C03659=1172.172,406.681,-85.424,-176.064,9.284,148.745
C03660=1172.175,406.433,-85.388,-176.064,9.282,148.745
C03661=1172.179,406.186,-85.352,-176.063,9.280,148.744
C03662=1172.183,405.938,-85.316,-176.063,9.278,148.744
C03663=1172.187,405.691,-85.279,-176.062,9.276,148.743
C03664=1172.191,405.444,-85.244,-176.062,9.273,148.742
C03665=1172.195,405.197,-85.207,-176.062,9.272,148.742
C03666=1172.199,404.949,-85.171,-176.062,9.269,148.741
C03667=1172.204,404.702,-85.135,-176.062,9.267,148.740
C03668=1172.207,404.455,-85.099,-176.061,9.265,148.740
C03669=1172.211,404.207,-85.063,-176.061,9.263,148.739
C03670=1172.215,403.960,-85.027,-176.061,9.261,148.739
C03671=1172.219,403.713,-84.991,-176.060,9.259,148.738
C03672=1172.223,403.465,-84.955,-176.060,9.257,148.737
C03673=1172.226,403.218,-84.919,-176.060,9.255,148.737
C03674=1172.231,402.970,-84.883,-176.060,9.252,148.736
C03675=1172.234,402.724,-84.846,-176.059,9.250,148.735
C03676=1172.238,402.476,-84.810,-176.059,9.248,148.735
C03677=1172.242,402.228,-84.775,-176.059,9.245,148.734
C03678=1172.246,401.981,-84.738,-176.059,9.244,148.733
C03679=1172.250,401.734,-84.702,-176.058,9.241,148.733
C03680=1172.254,401.486,-84.665,-176.058,9.239,148.732
C03681=1172.258,401.239,-84.630,-176.058,9.237,148.731
C03682=1172.261,400.991,-84.594,-176.057,9.234,148.731
C03683=1172.266,400.745,-84.558,-176.058,9.232,148.730
C03684=1172.270,400.497,-84.522,-176.057,9.230,148.729
C03685=1172.274,400.250,-84.486,-176.057,9.228,148.729
C03686=1172.277,400.003,-84.450,-176.057,9.225,148.728
C03687=1172.282,399.755,-84.414,-176.056,9.222,148.727
C03688=1172.285,399.507,-84.378,-176.056,9.220,148.727
C03689=1172.289,399.260,-84.342,-176.056,9.218,148.726
C03690=1172.293,399.013,-84.306,-176.056,9.216,148.725
C03691=1172.297,398.765,-84.270,-176.056,9.213,148.725
C03692=1172.301,398.518,-84.233,-176.056,9.211,148.724
C03693=1172.305,398.270,-84.198,-176.055,9.208,148.723
C03694=1172.308,398.023,-84.162,-176.055,9.206,148.723
C03695=1172.313,397.776,-84.126,-176.055,9.204,148.722
C03696=1172.317,397.529,-84.090,-176.054,9.201,148.721
C03697=1172.321,397.281,-84.054,-176.054,9.199,148.720
C03698=1172.324,397.034,-84.018,-176.054,9.196,148.720
C03699=1172.328,396.787,-83.982,-176.054,9.194,148.719
C03700=1172.332,396.539,-83.946,-176.054,9.191,148.718
C03701=1172.336,396.291,-83.911,-176.054,9.189,148.718
C03702=1172.340,396.044,-83.874,-176.054,9.186,148.717
C03703=1172.344,395.797,-83.838,-176.054,9.184,148.716
C03704=1172.347,395.549,-83.803,-176.054,9.181,148.716
C03705=1172.352,395.303,-83.766,-176.053,9.179,148.715
C03706=1172.356,395.055,-83.731,-176.053,9.176,148.714
C03707=1172.360,394.807,-83.694,-176.053,9.173,148.713
C03708=1172.364,394.560,-83.659,-176.053,9.171,148.713
C03709=1172.367,394.313,-83.623,-176.053,9.167,148.712
C03710=1172.372,394.065,-83.587,-176.053,9.165,148.711
C03711=1172.375,393.818,-83.551,-176.053,9.162,148.711
C03712=1172.379,393.570,-83.515,-176.053,9.160,148.710
C03713=1172.383,393.323,-83.479,-176.053,9.157,148.709
C03714=1172.387,393.076,-83.443,-176.053,9.155,148.709
C03715=1172.391,392.829,-83.408,-176.053,9.152,148.708
C03716=1172.395,392.581,-83.372,-176.053,9.149,148.707
C03717=1172.399,392.334,-83.335,-176.053,9.146,148.706
C03718=1172.404,392.049,-83.294,-176.053,9.143,148.705
C03719=1172.408,391.765,-83.253,-176.053,9.140,148.705
C03720=1172.412,391.480,-83.212,-176.053,9.137,148.704
C03721=1172.417,391.195,-83.171,-176.053,9.133,148.703
C03722=1172.421,390.948,-83.135,-176.054,9.131,148.702
C03723=1172.425,390.700,-83.099,-176.054,9.127,148.702
C03724=1172.429,390.453,-83.063,-176.054,9.125,148.701
C03725=1172.432,390.205,-83.028,-176.054,9.121,148.700
C03726=1172.437,389.957,-82.992,-176.054,9.119,148.699
C03727=1172.440,389.711,-82.955,-176.055,9.115,148.699
C03728=1172.444,389.463,-82.920,-176.054,9.113,148.698
C03729=1172.449,389.216,-82.884,-176.055,9.110,148.697
C03730=1172.452,388.968,-82.848,-176.055,9.107,148.697
C03731=1172.456,388.721,-82.813,-176.055,9.104,148.696
C03732=1172.460,388.473,-82.777,-176.055,9.101,148.695
C03733=1172.464,388.226,-82.741,-176.056,9.098,148.694
C03734=1172.468,387.978,-82.706,-176.057,9.095,148.694
C03735=1172.472,387.732,-82.670,-176.056,9.092,148.693
C03736=1172.475,387.484,-82.634,-176.057,9.089,148.692
C03737=1172.480,387.237,-82.598,-176.057,9.085,148.692
C03738=1172.483,386.989,-82.562,-176.058,9.082,148.691
C03739=1172.487,386.742,-82.527,-176.058,9.080,148.690
C03740=1172.491,386.494,-82.491,-176.058,9.076,148.690
C03741=1172.496,386.247,-82.456,-176.059,9.073,148.689
C03742=1172.499,386.000,-82.420,-176.060,9.070,148.688
C03743=1172.503,385.752,-82.385,-176.060,9.067,148.687
C03744=1172.507,385.505,-82.349,-176.061,9.063,148.687
C03745=1172.511,385.257,-82.313,-176.061,9.060,148.686
C03746=1172.515,385.009,-82.277,-176.062,9.057,148.685
C03747=1172.519,384.762,-82.242,-176.062,9.054,148.685
C03748=1172.523,384.515,-82.207,-176.063,9.050,148.684
C03749=1172.526,384.267,-82.171,-176.064,9.047,148.683
C03750=1172.531,384.020,-82.135,-176.064,9.044,148.683
C03751=1172.534,383.772,-82.099,-176.065,9.041,148.682
C03752=1172.539,383.525,-82.064,-176.065,9.037,148.681
C03753=1172.542,383.278,-82.029,-176.066,9.034,148.681
C03754=1172.546,383.030,-81.993,-176.067,9.031,148.680
C03755=1172.550,382.782,-81.957,-176.067,9.028,148.679
C03756=1172.555,382.536,-81.922,-176.068,9.025,148.679
C03757=1172.558,382.288,-81.886,-176.069,9.020,148.678
C03758=1172.562,382.041,-81.851,-176.070,9.017,148.677
C03759=1172.566,381.793,-81.815,-176.071,9.014,148.677
C03760=1172.569,381.546,-81.780,-176.071,9.011,148.676
C03761=1172.574,381.299,-81.744,-176.073,9.007,148.675
C03762=1172.578,381.051,-81.708,-176.074,9.004,148.675
C03763=1172.582,380.804,-81.673,-176.074,9.000,148.674
C03764=1172.586,380.555,-81.638,-176.075,8.997,148.673
C03765=1172.590,380.309,-81.603,-176.076,8.993,148.673
C03766=1172.594,380.061,-81.567,-176.077,8.990,148.672
C03767=1172.597,379.814,-81.532,-176.078,8.986,148.671
C03768=1172.602,379.566,-81.495,-176.079,8.983,148.671
C03769=1172.606,379.319,-81.460,-176.080,8.980,148.670
C03770=1172.610,379.072,-81.425,-176.081,8.976,148.670
C03771=1172.614,378.823,-81.390,-176.082,8.973,148.669
C03772=1172.618,378.577,-81.355,-176.083,8.969,148.668
C03773=1172.621,378.329,-81.319,-176.084,8.966,148.668
C03774=1172.625,378.082,-81.284,-176.086,8.962,148.667
C03775=1172.629,377.834,-81.249,-176.087,8.959,148.667
C03776=1172.633,377.587,-81.214,-176.088,8.955,148.666
C03777=1172.637,377.339,-81.178,-176.089,8.951,148.665
C03778=1172.641,377.092,-81.142,-176.090,8.948,148.665
C03779=1172.645,376.844,-81.108,-176.092,8.944,148.664
C03780=1172.649,376.597,-81.072,-176.092,8.941,148.664
C03781=1172.653,376.349,-81.037,-176.094,8.937,148.663
C03782=1172.657,376.103,-81.002,-176.095,8.933,148.662
C03783=1172.661,375.854,-80.967,-176.097,8.930,148.662
C03784=1172.664,375.607,-80.931,-176.098,8.926,148.661
C03785=1172.668,375.359,-80.896,-176.099,8.923,148.661
C03786=1172.673,375.112,-80.861,-176.100,8.919,148.660
C03787=1172.676,374.864,-80.826,-176.102,8.916,148.660
C03788=1172.680,374.617,-80.790,-176.103,8.912,148.659
C03789=1172.685,374.370,-80.756,-176.105,8.908,148.658
C03790=1172.688,374.122,-80.720,-176.106,8.905,148.658
C03791=1172.692,373.874,-80.685,-176.108,8.901,148.657
C03792=1172.696,373.627,-80.650,-176.109,8.897,148.657
C03793=1172.700,373.380,-80.615,-176.111,8.894,148.656
C03794=1172.705,373.132,-80.580,-176.112,8.890,148.656
C03795=1172.708,372.885,-80.545,-176.114,8.886,148.655
C03796=1172.712,372.637,-80.510,-176.115,8.883,148.655
C03797=1172.717,372.390,-80.475,-176.117,8.880,148.654
C03798=1172.721,372.142,-80.440,-176.118,8.876,148.654
C03799=1172.724,371.894,-80.404,-176.120,8.872,148.653
C03800=1172.729,371.647,-80.370,-176.121,8.868,148.653
C03801=1172.732,371.400,-80.335,-176.123,8.864,148.652
C03802=1172.736,371.152,-80.300,-176.125,8.861,148.651
C03803=1172.740,370.905,-80.265,-176.126,8.857,148.651
C03804=1172.744,370.656,-80.230,-176.128,8.853,148.651
C03805=1172.748,370.410,-80.195,-176.130,8.849,148.650
C03806=1172.752,370.162,-80.160,-176.132,8.846,148.650
C03807=1172.757,369.914,-80.125,-176.133,8.842,148.649
C03808=1172.760,369.667,-80.090,-176.135,8.839,148.649
C03809=1172.764,369.419,-80.056,-176.137,8.835,148.648
C03810=1172.768,369.172,-80.021,-176.138,8.831,148.648
C03811=1172.772,368.924,-79.986,-176.140,8.827,148.647
C03812=1172.776,368.677,-79.951,-176.142,8.824,148.647
C03813=1172.780,368.429,-79.916,-176.144,8.820,148.646
C03814=1172.784,368.182,-79.882,-176.146,8.817,148.646
C03815=1172.788,367.934,-79.847,-176.148,8.813,148.646
C03816=1172.792,367.686,-79.811,-176.150,8.809,148.645
C03817=1172.796,367.439,-79.777,-176.151,8.806,148.645
C03818=1172.800,367.191,-79.742,-176.153,8.802,148.644
C03819=1172.804,366.944,-79.708,-176.155,8.799,148.644
C03820=1172.808,366.696,-79.673,-176.157,8.795,148.643
C03821=1172.812,366.449,-79.638,-176.159,8.791,148.643
C03822=1172.816,366.166,-79.598,-176.161,8.787,148.642
C03823=1172.821,365.885,-79.559,-176.164,8.783,148.642
C03824=1172.825,365.603,-79.520,-176.166,8.778,148.641
C03825=1172.830,365.321,-79.480,-176.168,8.774,148.641
C03826=1172.834,365.073,-79.445,-176.170,8.771,148.641
C03827=1172.838,364.826,-79.411,-176.172,8.766,148.640
C03828=1172.842,364.578,-79.377,-176.174,8.763,148.640
C03829=1172.846,364.330,-79.342,-176.176,8.759,148.639
C03830=1172.850,364.082,-79.307,-176.178,8.756,148.639
C03831=1172.854,363.835,-79.274,-176.180,8.752,148.639
C03832=1172.858,363.588,-79.238,-176.182,8.748,148.638
C03833=1172.861,363.340,-79.204,-176.185,8.745,148.638
C03834=1172.866,363.093,-79.170,-176.186,8.741,148.638
C03835=1172.870,362.845,-79.135,-176.188,8.737,148.637
C03836=1172.874,362.598,-79.101,-176.191,8.734,148.637
C03837=1172.878,362.350,-79.066,-176.193,8.730,148.636
C03838=1172.882,362.103,-79.032,-176.195,8.726,148.636
C03839=1172.886,361.854,-78.997,-176.197,8.723,148.636
C03840=1172.890,361.607,-78.963,-176.199,8.719,148.635
C03841=1172.893,361.359,-78.929,-176.201,8.716,148.635
C03842=1172.898,361.112,-78.894,-176.204,8.711,148.635
C03843=1172.902,360.865,-78.860,-176.206,8.708,148.634
C03844=1172.906,360.617,-78.826,-176.208,8.704,148.634
C03845=1172.910,360.369,-78.792,-176.210,8.701,148.634
C03846=1172.913,360.121,-78.757,-176.212,8.697,148.633
C03847=1172.918,359.874,-78.724,-176.215,8.693,148.633
C03848=1172.922,359.626,-78.689,-176.217,8.690,148.633
C03849=1172.925,359.378,-78.655,-176.219,8.686,148.632
C03850=1172.930,359.131,-78.621,-176.221,8.682,148.632
C03851=1172.933,358.883,-78.586,-176.223,8.679,148.632
C03852=1172.938,358.636,-78.552,-176.225,8.675,148.631
C03853=1172.942,358.388,-78.519,-176.228,8.672,148.631
C03854=1172.946,358.140,-78.484,-176.230,8.668,148.631
C03855=1172.950,357.893,-78.450,-176.232,8.664,148.630
C03856=1172.954,357.645,-78.416,-176.235,8.661,148.630
C03857=1172.958,357.398,-78.381,-176.237,8.657,148.630
C03858=1172.962,357.149,-78.348,-176.239,8.653,148.629
C03859=1172.966,356.902,-78.314,-176.242,8.650,148.629
C03860=1172.969,356.655,-78.279,-176.244,8.646,148.629
C03861=1172.974,356.407,-78.245,-176.246,8.643,148.629
C03862=1172.978,356.159,-78.212,-176.248,8.640,148.628
C03863=1172.982,355.911,-78.177,-176.251,8.635,148.628
C03864=1172.986,355.664,-78.143,-176.253,8.632,148.628
C03865=1172.990,355.416,-78.110,-176.255,8.628,148.627
C03866=1172.994,355.168,-78.075,-176.257,8.625,148.627
C03867=1172.998,354.921,-78.042,-176.260,8.621,148.627
C03868=1173.002,354.674,-78.008,-176.262,8.617,148.627
C03869=1173.007,354.426,-77.974,-176.264,8.614,148.626
C03870=1173.010,354.178,-77.940,-176.266,8.611,148.626
C03871=1173.014,353.931,-77.906,-176.269,8.607,148.626
C03872=1173.019,353.683,-77.872,-176.271,8.603,148.625
C03873=1173.023,353.435,-77.839,-176.273,8.600,148.625
C03874=1173.026,353.187,-77.805,-176.276,8.597,148.625
C03875=1173.031,352.940,-77.771,-176.278,8.593,148.625
C03876=1173.035,352.692,-77.737,-176.281,8.589,148.624
C03877=1173.039,352.445,-77.704,-176.283,8.585,148.624
C03878=1173.042,352.196,-77.670,-176.285,8.582,148.624
C03879=1173.047,351.949,-77.636,-176.287,8.579,148.624
C03880=1173.051,351.701,-77.602,-176.289,8.576,148.623
C03881=1173.055,351.454,-77.569,-176.292,8.571,148.623
C03882=1173.058,351.206,-77.535,-176.295,8.568,148.623
C03883=1173.063,350.958,-77.501,-176.296,8.565,148.622
C03884=1173.067,350.710,-77.467,-176.299,8.561,148.622
C03885=1173.071,350.463,-77.434,-176.301,8.558,148.622
C03886=1173.075,350.216,-77.400,-176.304,8.554,148.622
C03887=1173.079,349.967,-77.367,-176.306,8.550,148.622
C03888=1173.083,349.719,-77.333,-176.308,8.547,148.621
C03889=1173.087,349.472,-77.299,-176.311,8.544,148.621
C03890=1173.091,349.224,-77.266,-176.313,8.541,148.621
C03891=1173.096,348.977,-77.233,-176.315,8.536,148.620
C03892=1173.099,348.729,-77.199,-176.318,8.533,148.620
C03893=1173.103,348.481,-77.166,-176.320,8.530,148.620
C03894=1173.108,348.233,-77.132,-176.322,8.526,148.620
C03895=1173.112,347.985,-77.099,-176.324,8.523,148.620
C03896=1173.116,347.738,-77.065,-176.327,8.519,148.619
C03897=1173.120,347.490,-77.032,-176.330,8.515,148.619
C03898=1173.124,347.243,-76.998,-176.332,8.512,148.619
C03899=1173.128,346.995,-76.965,-176.334,8.509,148.619
C03900=1173.132,346.747,-76.932,-176.336,8.506,148.618
C03901=1173.136,346.499,-76.898,-176.339,8.502,148.618
C03902=1173.140,346.252,-76.865,-176.342,8.498,148.618
C03903=1173.144,346.004,-76.832,-176.344,8.495,148.618
C03904=1173.148,345.756,-76.798,-176.346,8.492,148.618
C03905=1173.153,345.508,-76.765,-176.348,8.488,148.617
C03906=1173.157,345.260,-76.732,-176.351,8.485,148.617
C03907=1173.161,345.013,-76.698,-176.353,8.482,148.617
C03908=1173.165,344.765,-76.665,-176.356,8.478,148.617
C03909=1173.169,344.517,-76.632,-176.358,8.474,148.616
C03910=1173.174,344.270,-76.599,-176.360,8.471,148.616
C03911=1173.178,344.022,-76.566,-176.363,8.468,148.616
C03912=1173.181,343.773,-76.532,-176.365,8.464,148.616
C03913=1173.185,343.526,-76.499,-176.367,8.461,148.616
C03914=1173.190,343.278,-76.466,-176.370,8.457,148.615
C03915=1173.194,343.030,-76.433,-176.372,8.454,148.615
C03916=1173.198,342.782,-76.400,-176.375,8.450,148.615
C03917=1173.201,342.535,-76.367,-176.377,8.447,148.615
C03918=1173.205,342.287,-76.334,-176.379,8.444,148.614
C03919=1173.209,342.040,-76.301,-176.382,8.441,148.614
C03920=1173.214,341.792,-76.268,-176.384,8.437,148.614
C03921=1173.218,341.544,-76.234,-176.387,8.433,148.614
C03922=1173.222,341.296,-76.201,-176.389,8.430,148.614
C03923=1173.226,341.049,-76.168,-176.392,8.427,148.614
C03924=1173.230,340.801,-76.135,-176.394,8.423,148.613
C03925=1173.235,340.553,-76.103,-176.396,8.420,148.613
C03926=1173.239,340.274,-76.066,-176.399,8.416,148.613
C03927=1173.244,339.994,-76.028,-176.402,8.412,148.613
C03928=1173.248,339.715,-75.991,-176.405,8.409,148.613
C03929=1173.253,339.436,-75.954,-176.407,8.405,148.612
C03930=1173.257,339.189,-75.921,-176.410,8.401,148.612
C03931=1173.261,338.940,-75.889,-176.412,8.398,148.612
C03932=1173.265,338.693,-75.856,-176.414,8.395,148.612
C03933=1173.270,338.445,-75.822,-176.416,8.391,148.612
C03934=1173.273,338.197,-75.790,-176.419,8.388,148.612
C03935=1173.277,337.949,-75.757,-176.422,8.384,148.611
C03936=1173.282,337.701,-75.724,-176.424,8.381,148.611
C03937=1173.286,337.454,-75.691,-176.427,8.378,148.611
C03938=1173.289,337.206,-75.659,-176.429,8.374,148.611
C03939=1173.294,336.958,-75.626,-176.431,8.371,148.610
C03940=1173.298,336.709,-75.594,-176.434,8.368,148.610
C03941=1173.303,336.462,-75.561,-176.436,8.365,148.610
C03942=1173.306,336.215,-75.528,-176.438,8.362,148.610
C03943=1173.311,335.967,-75.496,-176.441,8.357,148.610
C03944=1173.315,335.719,-75.463,-176.444,8.354,148.610
C03945=1173.318,335.471,-75.431,-176.446,8.351,148.610
C03946=1173.323,335.223,-75.398,-176.449,8.348,148.609
C03947=1173.327,334.975,-75.365,-176.451,8.344,148.609
C03948=1173.331,334.727,-75.332,-176.453,8.341,148.609
C03949=1173.335,334.480,-75.300,-176.456,8.338,148.609
C03950=1173.340,334.232,-75.267,-176.458,8.335,148.609
C03951=1173.343,333.985,-75.235,-176.460,8.332,148.609
C03952=1173.347,333.736,-75.202,-176.463,8.327,148.608
C03953=1173.352,333.488,-75.170,-176.466,8.324,148.608
C03954=1173.355,333.240,-75.137,-176.468,8.321,148.608
C03955=1173.360,332.992,-75.105,-176.471,8.318,148.608
C03956=1173.364,332.744,-75.072,-176.473,8.315,148.608
C03957=1173.368,332.497,-75.040,-176.476,8.312,148.608
C03958=1173.373,332.249,-75.008,-176.478,8.308,148.607
C03959=1173.376,332.001,-74.975,-176.480,8.305,148.607
C03960=1173.380,331.753,-74.943,-176.483,8.302,148.607
C03961=1173.384,331.506,-74.910,-176.485,8.299,148.607
C03962=1173.389,331.258,-74.878,-176.487,8.295,148.607
C03963=1173.393,331.010,-74.846,-176.491,8.292,148.607
C03964=1173.397,330.762,-74.813,-176.493,8.288,148.607
C03965=1173.401,330.514,-74.781,-176.495,8.285,148.606
C03966=1173.405,330.266,-74.749,-176.498,8.282,148.606
C03967=1173.410,330.018,-74.717,-176.500,8.279,148.606
C03968=1173.413,329.771,-74.684,-176.503,8.275,148.606
C03969=1173.418,329.522,-74.652,-176.505,8.272,148.606
C03970=1173.421,329.274,-74.620,-176.508,8.269,148.606
C03971=1173.427,329.027,-74.588,-176.510,8.266,148.606
C03972=1173.430,328.779,-74.556,-176.513,8.263,148.606
C03973=1173.434,328.531,-74.523,-176.515,8.259,148.605
C03974=1173.438,328.283,-74.491,-176.517,8.256,148.605
C03975=1173.442,328.035,-74.460,-176.520,8.252,148.605
C03976=1173.447,327.787,-74.427,-176.523,8.249,148.605
C03977=1173.451,327.539,-74.395,-176.525,8.246,148.605
C03978=1173.455,327.291,-74.363,-176.528,8.243,148.605
C03979=1173.459,327.043,-74.332,-176.530,8.239,148.605
C03980=1173.463,326.796,-74.299,-176.532,8.236,148.604
C03981=1173.467,326.548,-74.267,-176.535,8.233,148.604
C03982=1173.471,326.300,-74.235,-176.537,8.230,148.604
C03983=1173.476,326.052,-74.203,-176.540,8.227,148.604
C03984=1173.480,325.804,-74.171,-176.542,8.224,148.604
C03985=1173.484,325.557,-74.139,-176.544,8.220,148.604
C03986=1173.488,325.308,-74.107,-176.547,8.217,148.604
C03987=1173.492,325.060,-74.075,-176.549,8.214,148.604
C03988=1173.496,324.812,-74.043,-176.552,8.211,148.604
C03989=1173.501,324.564,-74.011,-176.554,8.208,148.603
C03990=1173.505,324.316,-73.979,-176.557,8.204,148.603
C03991=1173.508,324.068,-73.947,-176.560,8.201,148.603
C03992=1173.513,323.821,-73.916,-176.562,8.197,148.603
C03993=1173.517,323.572,-73.884,-176.565,8.194,148.603
C03994=1173.522,323.325,-73.853,-176.567,8.191,148.603
C03995=1173.525,323.077,-73.821,-176.570,8.188,148.603
C03996=1173.530,322.828,-73.788,-176.572,8.185,148.602
C03997=1173.534,322.581,-73.757,-176.575,8.181,148.602
C03998=1173.538,322.333,-73.725,-176.577,8.178,148.602
C03999=1173.541,322.085,-73.693,-176.580,8.175,148.602
C04000=1173.546,321.837,-73.662,-176.582,8.172,148.602
C04001=1173.551,321.589,-73.630,-176.585,8.169,148.602
C04002=1173.555,321.341,-73.599,-176.587,8.166,148.602
C04003=1173.559,321.093,-73.567,-176.590,8.163,148.602
C04004=1173.562,320.845,-73.535,-176.592,8.160,148.602
C04005=1173.567,320.597,-73.504,-176.595,8.156,148.602
C04006=1173.571,320.349,-73.472,-176.597,8.153,148.602
C04007=1173.576,320.102,-73.440,-176.600,8.150,148.601
C04008=1173.579,319.854,-73.408,-176.602,8.147,148.601
C04009=1173.583,319.605,-73.377,-176.605,8.144,148.601
C04010=1173.588,319.358,-73.346,-176.607,8.141,148.601
C04011=1173.591,319.109,-73.314,-176.610,8.137,148.601
C04012=1173.596,318.862,-73.283,-176.612,8.134,148.601
C04013=1173.600,318.613,-73.251,-176.615,8.131,148.601
C04014=1173.605,318.366,-73.219,-176.617,8.128,148.601
C04015=1173.609,318.117,-73.188,-176.620,8.125,148.601
C04016=1173.613,317.870,-73.157,-176.622,8.122,148.601
C04017=1173.617,317.621,-73.125,-176.625,8.118,148.600
C04018=1173.621,317.374,-73.094,-176.628,8.115,148.600
C04019=1173.625,317.126,-73.062,-176.630,8.111,148.600
C04020=1173.630,316.878,-73.031,-176.633,8.108,148.600
C04021=1173.633,316.630,-73.000,-176.635,8.105,148.600
C04022=1173.638,316.382,-72.969,-176.638,8.102,148.600
C04023=1173.642,316.134,-72.937,-176.640,8.099,148.600
C04024=1173.646,315.886,-72.906,-176.643,8.096,148.600
C04025=1173.650,315.638,-72.874,-176.645,8.093,148.600
C04026=1173.655,315.390,-72.844,-176.648,8.090,148.600
C04027=1173.658,315.142,-72.812,-176.650,8.086,148.599
C04028=1173.663,314.894,-72.781,-176.653,8.083,148.599
C04029=1173.667,314.645,-72.750,-176.655,8.080,148.599
C04030=1173.672,314.368,-72.715,-176.658,8.077,148.599
C04031=1173.676,314.092,-72.680,-176.661,8.073,148.599
C04032=1173.681,313.815,-72.645,-176.664,8.070,148.599
C04033=1173.686,313.538,-72.610,-176.667,8.066,148.599
C04034=1173.690,313.291,-72.579,-176.670,8.063,148.599
C04035=1173.694,313.042,-72.548,-176.672,8.060,148.599
C04036=1173.698,312.794,-72.517,-176.675,8.057,148.599
C04037=1173.702,312.546,-72.486,-176.677,8.053,148.599
C04038=1173.707,312.298,-72.455,-176.680,8.050,148.599
C04039=1173.711,312.050,-72.424,-176.682,8.047,148.598
C04040=1173.715,311.802,-72.392,-176.685,8.044,148.599
C04041=1173.720,311.554,-72.361,-176.687,8.041,148.599
C04042=1173.724,311.305,-72.330,-176.690,8.038,148.598
C04043=1173.728,311.058,-72.300,-176.692,8.035,148.598
C04044=1173.732,310.810,-72.269,-176.695,8.032,148.598
C04045=1173.736,310.562,-72.237,-176.697,8.029,148.598
C04046=1173.740,310.314,-72.207,-176.700,8.026,148.598
C04047=1173.745,310.066,-72.176,-176.702,8.023,148.598
C04048=1173.749,309.817,-72.145,-176.705,8.020,148.598
C04049=1173.753,309.570,-72.115,-176.707,8.017,148.598
C04050=1173.757,309.321,-72.083,-176.710,8.014,148.598
C04051=1173.761,309.074,-72.052,-176.712,8.011,148.598
C04052=1173.766,308.826,-72.021,-176.715,8.008,148.598
C04053=1173.770,308.577,-71.990,-176.717,8.005,148.598
C04054=1173.774,308.329,-71.960,-176.720,8.001,148.598
C04055=1173.778,308.081,-71.929,-176.722,7.998,148.598
C04056=1173.782,307.833,-71.898,-176.725,7.995,148.598
C04057=1173.787,307.585,-71.867,-176.727,7.992,148.597
C04058=1173.791,307.337,-71.837,-176.730,7.989,148.597
C04059=1173.796,307.089,-71.806,-176.733,7.986,148.597
C04060=1173.800,306.840,-71.775,-176.735,7.983,148.597
C04061=1173.804,306.592,-71.745,-176.738,7.980,148.597
C04062=1173.808,306.345,-71.714,-176.741,7.977,148.597
C04063=1173.812,306.096,-71.683,-176.743,7.974,148.597
C04064=1173.817,305.848,-71.652,-176.746,7.971,148.597
C04065=1173.821,305.601,-71.622,-176.748,7.968,148.597
C04066=1173.825,305.353,-71.592,-176.751,7.964,148.597
C04067=1173.829,305.104,-71.560,-176.753,7.961,148.597
C04068=1173.833,304.856,-71.530,-176.756,7.958,148.597
C04069=1173.838,304.608,-71.499,-176.758,7.955,148.597
C04070=1173.842,304.360,-71.469,-176.761,7.952,148.597
C04071=1173.846,304.111,-71.439,-176.764,7.949,148.597
C04072=1173.850,303.863,-71.408,-176.766,7.946,148.597
C04073=1173.854,303.616,-71.378,-176.769,7.943,148.597
C04074=1173.859,303.368,-71.347,-176.772,7.940,148.597
C04075=1173.864,303.120,-71.316,-176.774,7.936,148.597
C04076=1173.867,302.872,-71.286,-176.777,7.933,148.597
C04077=1173.872,302.623,-71.256,-176.779,7.931,148.597
C04078=1173.876,302.375,-71.226,-176.781,7.928,148.596
C04079=1173.880,302.127,-71.195,-176.784,7.925,148.596
C04080=1173.885,301.879,-71.164,-176.786,7.922,148.596
C04081=1173.888,301.630,-71.134,-176.789,7.919,148.596
C04082=1173.893,301.382,-71.104,-176.791,7.916,148.596
C04083=1173.897,301.135,-71.073,-176.794,7.913,148.596
C04084=1173.902,300.886,-71.043,-176.797,7.910,148.596
C04085=1173.906,300.639,-71.013,-176.799,7.907,148.596
C04086=1173.910,300.390,-70.982,-176.802,7.904,148.596
C04087=1173.914,300.142,-70.953,-176.805,7.901,148.596
C04088=1173.918,299.894,-70.922,-176.807,7.897,148.596
C04089=1173.922,299.646,-70.892,-176.810,7.894,148.596
C04090=1173.927,299.397,-70.862,-176.812,7.891,148.596
C04091=1173.931,299.150,-70.831,-176.815,7.888,148.596
C04092=1173.935,298.902,-70.802,-176.817,7.885,148.596
C04093=1173.939,298.653,-70.771,-176.820,7.883,148.596
C04094=1173.943,298.405,-70.741,-176.822,7.880,148.596
C04095=1173.948,298.157,-70.711,-176.825,7.877,148.596
C04096=1173.952,297.909,-70.680,-176.827,7.874,148.596
C04097=1173.957,297.660,-70.650,-176.830,7.871,148.596
C04098=1173.961,297.413,-70.620,-176.833,7.868,148.596
C04099=1173.965,297.165,-70.591,-176.836,7.865,148.596
C04100=1173.970,296.917,-70.560,-176.838,7.861,148.596
C04101=1173.974,296.668,-70.531,-176.841,7.858,148.596
C04102=1173.978,296.421,-70.500,-176.843,7.855,148.596
C04103=1173.982,296.171,-70.470,-176.846,7.852,148.596
C04104=1173.986,295.923,-70.441,-176.848,7.849,148.596
C04105=1173.990,295.675,-70.410,-176.851,7.846,148.596
C04106=1173.995,295.427,-70.380,-176.853,7.844,148.596
C04107=1173.999,295.179,-70.350,-176.856,7.841,148.596
C04108=1174.003,294.931,-70.321,-176.858,7.838,148.596
C04109=1174.008,294.682,-70.291,-176.861,7.835,148.596
C04110=1174.012,294.435,-70.260,-176.864,7.832,148.596
C04111=1174.016,294.186,-70.231,-176.866,7.829,148.596
C04112=1174.020,293.938,-70.202,-176.869,7.825,148.595
C04113=1174.025,293.690,-70.171,-176.871,7.822,148.596
C04114=1174.029,293.442,-70.141,-176.874,7.819,148.596
C04115=1174.033,293.194,-70.112,-176.877,7.817,148.596
C04116=1174.037,292.946,-70.082,-176.879,7.814,148.596
C04117=1174.042,292.698,-70.052,-176.881,7.811,148.595
C04118=1174.046,292.449,-70.022,-176.884,7.808,148.596
C04119=1174.050,292.201,-69.993,-176.887,7.805,148.596
C04120=1174.055,291.953,-69.963,-176.890,7.802,148.596
C04121=1174.058,291.705,-69.933,-176.892,7.799,148.596
C04122=1174.063,291.456,-69.903,-176.895,7.796,148.595
C04123=1174.067,291.208,-69.874,-176.897,7.793,148.595
C04124=1174.072,290.960,-69.844,-176.900,7.790,148.595
C04125=1174.076,290.712,-69.815,-176.903,7.787,148.596
C04126=1174.080,290.463,-69.785,-176.905,7.785,148.596
C04127=1174.084,290.216,-69.755,-176.908,7.782,148.596
C04128=1174.089,289.967,-69.725,-176.910,7.778,148.595
C04129=1174.093,289.719,-69.696,-176.913,7.775,148.595
C04130=1174.097,289.471,-69.666,-176.915,7.773,148.596
C04131=1174.101,289.222,-69.637,-176.918,7.770,148.596
C04132=1174.106,288.974,-69.607,-176.921,7.767,148.596
C04133=1174.110,288.726,-69.578,-176.923,7.763,148.595
C04134=1174.115,288.452,-69.545,-176.926,7.760,148.595
C04135=1174.119,288.177,-69.513,-176.929,7.757,148.595
C04136=1174.124,287.901,-69.480,-176.931,7.754,148.595
C04137=1174.129,287.627,-69.447,-176.935,7.751,148.595
C04138=1174.134,287.379,-69.418,-176.937,7.748,148.596
C04139=1174.138,287.131,-69.388,-176.940,7.745,148.596
C04140=1174.142,286.882,-69.359,-176.942,7.742,148.596
C04141=1174.146,286.634,-69.329,-176.945,7.739,148.596
C04142=1174.150,286.386,-69.300,-176.947,7.736,148.595
C04143=1174.154,286.138,-69.271,-176.950,7.733,148.596
C04144=1174.159,285.889,-69.242,-176.953,7.730,148.596
C04145=1174.164,285.641,-69.213,-176.956,7.727,148.596
C04146=1174.168,285.393,-69.183,-176.958,7.725,148.596
C04147=1174.172,285.145,-69.154,-176.960,7.722,148.596
C04148=1174.176,284.896,-69.124,-176.963,7.719,148.596
C04149=1174.180,284.648,-69.095,-176.966,7.716,148.596
C04150=1174.185,284.399,-69.066,-176.968,7.713,148.596
C04151=1174.190,284.152,-69.037,-176.971,7.710,148.596
C04152=1174.194,283.903,-69.008,-176.974,7.707,148.596
C04153=1174.198,283.655,-68.978,-176.976,7.705,148.596
C04154=1174.202,283.407,-68.949,-176.979,7.702,148.596
C04155=1174.206,283.158,-68.921,-176.981,7.699,148.596
C04156=1174.210,282.910,-68.891,-176.984,7.696,148.596
C04157=1174.215,282.662,-68.862,-176.987,7.693,148.596
C04158=1174.219,282.414,-68.833,-176.990,7.690,148.596
C04159=1174.224,282.165,-68.804,-176.992,7.687,148.596
C04160=1174.228,281.917,-68.774,-176.994,7.684,148.596
C04161=1174.233,281.670,-68.745,-176.997,7.681,148.596
C04162=1174.237,281.421,-68.717,-176.999,7.678,148.596
C04163=1174.241,281.173,-68.688,-177.002,7.675,148.596
C04164=1174.245,280.924,-68.659,-177.005,7.672,148.596
C04165=1174.250,280.676,-68.630,-177.008,7.669,148.596
C04166=1174.254,280.428,-68.600,-177.010,7.667,148.596
C04167=1174.258,280.179,-68.572,-177.013,7.664,148.596
C04168=1174.263,279.931,-68.542,-177.015,7.661,148.596
C04169=1174.267,279.683,-68.514,-177.018,7.658,148.596
C04170=1174.271,279.435,-68.485,-177.021,7.655,148.596
C04171=1174.275,279.186,-68.456,-177.022,7.653,148.596
C04172=1174.280,278.937,-68.427,-177.025,7.650,148.596
C04173=1174.284,278.690,-68.398,-177.028,7.647,148.596
C04174=1174.288,278.441,-68.370,-177.031,7.644,148.596
C04175=1174.293,278.193,-68.340,-177.033,7.641,148.596
C04176=1174.297,277.944,-68.311,-177.036,7.638,148.596
C04177=1174.301,277.697,-68.283,-177.038,7.636,148.596
C04178=1174.306,277.448,-68.254,-177.041,7.633,148.596
C04179=1174.310,277.199,-68.225,-177.044,7.630,148.597
C04180=1174.314,276.952,-68.197,-177.047,7.627,148.597
C04181=1174.319,276.703,-68.168,-177.049,7.624,148.597
C04182=1174.323,276.455,-68.139,-177.051,7.622,148.597
C04183=1174.327,276.207,-68.111,-177.054,7.619,148.597
C04184=1174.332,275.958,-68.082,-177.057,7.616,148.597
C04185=1174.336,275.710,-68.053,-177.060,7.613,148.597
C04186=1174.340,275.462,-68.025,-177.062,7.610,148.597
C04187=1174.345,275.213,-67.996,-177.065,7.608,148.597
C04188=1174.349,274.965,-67.967,-177.067,7.605,148.597
C04189=1174.353,274.717,-67.939,-177.070,7.602,148.597
C04190=1174.358,274.468,-67.910,-177.073,7.599,148.597
C04191=1174.361,274.220,-67.881,-177.076,7.596,148.597
C04192=1174.366,273.972,-67.853,-177.078,7.594,148.597
C04193=1174.371,273.723,-67.824,-177.080,7.591,148.597
C04194=1174.375,273.475,-67.797,-177.083,7.588,148.597
C04195=1174.379,273.227,-67.767,-177.086,7.585,148.597
C04196=1174.383,272.978,-67.739,-177.089,7.582,148.597
C04197=1174.388,272.730,-67.711,-177.091,7.580,148.597
C04198=1174.392,272.481,-67.682,-177.094,7.577,148.598
C04199=1174.397,272.233,-67.654,-177.096,7.574,148.598
C04200=1174.400,271.985,-67.625,-177.099,7.571,148.598
C04201=1174.405,271.737,-67.597,-177.101,7.569,148.598
C04202=1174.409,271.489,-67.569,-177.104,7.566,148.598
C04203=1174.414,271.240,-67.540,-177.107,7.563,148.598
C04204=1174.418,270.992,-67.512,-177.109,7.560,148.598
C04205=1174.422,270.743,-67.483,-177.112,7.557,148.598
C04206=1174.427,270.495,-67.456,-177.114,7.555,148.598
C04207=1174.431,270.246,-67.427,-177.117,7.552,148.598
C04208=1174.435,269.999,-67.398,-177.120,7.549,148.598
C04209=1174.440,269.750,-67.370,-177.123,7.546,148.598
C04210=1174.444,269.502,-67.342,-177.125,7.544,148.598
C04211=1174.449,269.253,-67.313,-177.128,7.541,148.598
C04212=1174.453,269.005,-67.285,-177.130,7.538,148.598
C04213=1174.458,268.756,-67.257,-177.133,7.535,148.598
C04214=1174.462,268.509,-67.229,-177.135,7.532,148.598
C04215=1174.466,268.260,-67.201,-177.138,7.530,148.598
C04216=1174.471,268.012,-67.172,-177.141,7.527,148.599
C04217=1174.475,267.763,-67.145,-177.143,7.524,148.599
C04218=1174.480,267.514,-67.117,-177.146,7.521,148.599
C04219=1174.484,267.266,-67.088,-177.148,7.518,148.599
C04220=1174.488,267.018,-67.061,-177.151,7.515,148.599
C04221=1174.492,266.769,-67.032,-177.154,7.513,148.599
C04222=1174.497,266.521,-67.004,-177.156,7.510,148.599
C04223=1174.501,266.273,-66.976,-177.159,7.507,148.599
C04224=1174.506,266.024,-66.948,-177.161,7.504,148.599
C04225=1174.509,265.776,-66.920,-177.164,7.501,148.599
C04226=1174.514,265.527,-66.892,-177.167,7.500,148.599
C04227=1174.519,265.278,-66.864,-177.170,7.497,148.599
C04228=1174.523,265.031,-66.836,-177.172,7.494,148.599
C04229=1174.527,264.783,-66.808,-177.175,7.491,148.599
C04230=1174.531,264.534,-66.780,-177.177,7.489,148.600
C04231=1174.536,264.285,-66.752,-177.180,7.486,148.600
C04232=1174.540,264.037,-66.724,-177.183,7.483,148.600
C04233=1174.544,263.789,-66.696,-177.186,7.480,148.600
C04234=1174.550,263.541,-66.668,-177.188,7.478,148.600
C04235=1174.554,263.291,-66.641,-177.190,7.475,148.600
C04236=1174.558,263.044,-66.613,-177.193,7.472,148.600
C04237=1174.562,262.795,-66.585,-177.195,7.469,148.600
C04238=1174.567,262.522,-66.554,-177.199,7.467,148.600
C04239=1174.572,262.249,-66.524,-177.202,7.463,148.600
C04240=1174.576,261.976,-66.493,-177.205,7.460,148.600
C04241=1174.582,261.703,-66.463,-177.207,7.457,148.600
C04242=1174.586,261.454,-66.435,-177.210,7.455,148.601
C04243=1174.590,261.206,-66.408,-177.213,7.452,148.601
C04244=1174.594,260.958,-66.380,-177.215,7.449,148.601
C04245=1174.599,260.709,-66.352,-177.218,7.446,148.601
C04246=1174.603,260.461,-66.324,-177.220,7.444,148.601
C04247=1174.608,260.212,-66.297,-177.223,7.441,148.601
C04248=1174.612,259.964,-66.269,-177.226,7.438,148.601
C04249=1174.617,259.715,-66.242,-177.228,7.436,148.601
C04250=1174.621,259.467,-66.214,-177.231,7.433,148.601
C04251=1174.625,259.218,-66.186,-177.234,7.430,148.602
C04252=1174.629,258.970,-66.159,-177.236,7.428,148.602
C04253=1174.634,258.722,-66.132,-177.239,7.425,148.602
C04254=1174.638,258.473,-66.104,-177.242,7.422,148.602
C04255=1174.643,258.224,-66.076,-177.244,7.419,148.602
C04256=1174.647,257.977,-66.048,-177.247,7.417,148.602
C04257=1174.652,257.728,-66.021,-177.249,7.414,148.602
C04258=1174.656,257.479,-65.993,-177.253,7.412,148.602
C04259=1174.661,257.231,-65.966,-177.255,7.410,148.602
C04260=1174.665,256.982,-65.939,-177.257,7.407,148.602
C04261=1174.669,256.734,-65.911,-177.260,7.404,148.602
C04262=1174.674,256.485,-65.884,-177.262,7.401,148.602
C04263=1174.678,256.238,-65.856,-177.265,7.398,148.603
C04264=1174.683,255.989,-65.829,-177.268,7.396,148.603
C04265=1174.687,255.740,-65.801,-177.271,7.394,148.603
C04266=1174.691,255.492,-65.773,-177.273,7.391,148.603
C04267=1174.696,255.243,-65.746,-177.276,7.388,148.603
C04268=1174.700,254.995,-65.719,-177.278,7.386,148.603
C04269=1174.704,254.746,-65.692,-177.281,7.383,148.603
C04270=1174.709,254.498,-65.664,-177.284,7.380,148.603
C04271=1174.713,254.250,-65.638,-177.286,7.378,148.604
C04272=1174.717,254.001,-65.611,-177.289,7.375,148.604
C04273=1174.722,253.753,-65.584,-177.292,7.372,148.604
C04274=1174.726,253.504,-65.555,-177.294,7.370,148.604
C04275=1174.730,253.256,-65.528,-177.297,7.367,148.604
C04276=1174.735,253.007,-65.501,-177.300,7.364,148.604
C04277=1174.740,252.759,-65.474,-177.302,7.362,148.604
C04278=1174.744,252.510,-65.447,-177.305,7.359,148.604
C04279=1174.749,252.262,-65.420,-177.308,7.356,148.605
C04280=1174.752,252.013,-65.393,-177.310,7.354,148.605
C04281=1174.757,251.765,-65.366,-177.313,7.351,148.605
C04282=1174.761,251.516,-65.338,-177.316,7.348,148.605
C04283=1174.766,251.268,-65.311,-177.318,7.346,148.605
C04284=1174.771,251.019,-65.284,-177.321,7.344,148.605
C04285=1174.775,250.771,-65.257,-177.323,7.341,148.605
C04286=1174.779,250.522,-65.230,-177.326,7.338,148.605
C04287=1174.783,250.274,-65.203,-177.329,7.335,148.605
C04288=1174.788,250.025,-65.176,-177.331,7.334,148.606
C04289=1174.793,249.777,-65.149,-177.334,7.331,148.606
C04290=1174.797,249.528,-65.122,-177.337,7.328,148.606
C04291=1174.801,249.280,-65.096,-177.339,7.326,148.606
C04292=1174.806,249.031,-65.069,-177.342,7.323,148.606
C04293=1174.810,248.783,-65.042,-177.345,7.320,148.606
C04294=1174.815,248.534,-65.014,-177.347,7.318,148.606
C04295=1174.818,248.285,-64.988,-177.350,7.315,148.606
C04296=1174.823,248.037,-64.961,-177.353,7.313,148.607
C04297=1174.828,247.788,-64.934,-177.355,7.310,148.607
C04298=1174.832,247.540,-64.907,-177.358,7.307,148.607
C04299=1174.836,247.292,-64.880,-177.360,7.305,148.607
C04300=1174.841,247.043,-64.853,-177.364,7.302,148.607
C04301=1174.846,246.795,-64.826,-177.366,7.300,148.607
C04302=1174.850,246.546,-64.800,-177.369,7.297,148.607
C04303=1174.855,246.298,-64.773,-177.371,7.294,148.607
C04304=1174.859,246.049,-64.746,-177.374,7.292,148.608
C04305=1174.863,245.801,-64.720,-177.377,7.290,148.608
C04306=1174.868,245.552,-64.693,-177.379,7.287,148.608
C04307=1174.872,245.304,-64.665,-177.382,7.285,148.608
C04308=1174.877,245.055,-64.640,-177.385,7.282,148.608
C04309=1174.881,244.807,-64.613,-177.387,7.280,148.608
C04310=1174.885,244.558,-64.586,-177.390,7.277,148.608
C04311=1174.890,244.310,-64.559,-177.392,7.275,148.609
C04312=1174.895,244.061,-64.533,-177.395,7.272,148.609
C04313=1174.899,243.813,-64.506,-177.398,7.269,148.609
C04314=1174.903,243.564,-64.479,-177.401,7.267,148.609
C04315=1174.907,243.316,-64.453,-177.403,7.264,148.609
C04316=1174.912,243.067,-64.426,-177.405,7.262,148.609
C04317=1174.916,242.819,-64.400,-177.409,7.259,148.610
C04318=1174.921,242.570,-64.373,-177.411,7.256,148.610
C04319=1174.926,242.321,-64.347,-177.414,7.254,148.610
C04320=1174.930,242.073,-64.320,-177.417,7.252,148.610
C04321=1174.935,241.824,-64.294,-177.419,7.250,148.610
C04322=1174.939,241.575,-64.267,-177.422,7.247,148.610
C04323=1174.943,241.327,-64.240,-177.424,7.245,148.611
C04324=1174.948,241.078,-64.214,-177.427,7.242,148.611
C04325=1174.952,240.830,-64.187,-177.430,7.239,148.611
C04326=1174.956,240.581,-64.162,-177.433,7.237,148.611
C04327=1174.961,240.332,-64.135,-177.435,7.234,148.611
C04328=1174.965,240.084,-64.109,-177.437,7.232,148.611
C04329=1174.969,239.835,-64.082,-177.441,7.229,148.612
C04330=1174.974,239.587,-64.055,-177.443,7.227,148.612
C04331=1174.978,239.338,-64.030,-177.446,7.224,148.612
C04332=1174.983,239.090,-64.003,-177.449,7.222,148.612
C04333=1174.988,238.842,-63.977,-177.451,7.219,148.612
C04334=1174.993,238.592,-63.951,-177.454,7.216,148.612
C04335=1174.996,238.344,-63.924,-177.456,7.215,148.612
C04336=1175.001,238.095,-63.899,-177.459,7.212,148.613
C04337=1175.005,237.847,-63.872,-177.462,7.210,148.613
C04338=1175.010,237.598,-63.846,-177.465,7.207,148.613
C04339=1175.014,237.350,-63.819,-177.467,7.205,148.613
C04340=1175.018,237.101,-63.793,-177.470,7.202,148.613
C04341=1175.023,236.853,-63.768,-177.472,7.200,148.613
C04342=1175.028,236.581,-63.738,-177.475,7.197,148.614
C04343=1175.033,236.309,-63.710,-177.478,7.194,148.614
C04344=1175.037,236.038,-63.681,-177.481,7.192,148.614
C04345=1175.043,235.766,-63.653,-177.484,7.189,148.614
C04346=1175.047,235.518,-63.626,-177.486,7.187,148.614
C04347=1175.051,235.269,-63.601,-177.490,7.184,148.615
C04348=1175.057,235.020,-63.575,-177.492,7.182,148.615
C04349=1175.061,234.772,-63.548,-177.495,7.179,148.615
C04350=1175.065,234.523,-63.522,-177.498,7.176,148.615
C04351=1175.069,234.275,-63.497,-177.500,7.174,148.615
C04352=1175.074,234.025,-63.470,-177.503,7.172,148.615
C04353=1175.079,233.777,-63.445,-177.505,7.169,148.616
C04354=1175.083,233.529,-63.418,-177.508,7.167,148.616
C04355=1175.087,233.280,-63.393,-177.511,7.165,148.616
C04356=1175.092,233.031,-63.366,-177.514,7.162,148.616
C04357=1175.096,232.782,-63.341,-177.516,7.160,148.616
C04358=1175.101,232.534,-63.315,-177.519,7.157,148.616
C04359=1175.105,232.286,-63.289,-177.521,7.155,148.617
C04360=1175.110,232.037,-63.262,-177.524,7.152,148.617
C04361=1175.114,231.788,-63.237,-177.527,7.150,148.617
C04362=1175.119,231.540,-63.211,-177.530,7.147,148.617
C04363=1175.123,231.291,-63.185,-177.532,7.146,148.618
C04364=1175.127,231.042,-63.160,-177.535,7.143,148.618
C04365=1175.132,230.794,-63.134,-177.537,7.140,148.618
C04366=1175.137,230.545,-63.108,-177.540,7.138,148.618
C04367=1175.141,230.296,-63.082,-177.543,7.136,148.618
C04368=1175.146,230.048,-63.057,-177.546,7.133,148.618
C04369=1175.150,229.799,-63.031,-177.548,7.131,148.619
C04370=1175.155,229.551,-63.005,-177.551,7.128,148.619
C04371=1175.159,229.302,-62.980,-177.553,7.126,148.619
C04372=1175.163,229.053,-62.954,-177.557,7.124,148.619
C04373=1175.168,228.805,-62.928,-177.559,7.121,148.619
C04374=1175.173,228.556,-62.902,-177.562,7.119,148.620
C04375=1175.177,228.307,-62.876,-177.564,7.117,148.620
C04376=1175.182,228.059,-62.851,-177.567,7.115,148.620
C04377=1175.186,227.810,-62.825,-177.570,7.112,148.620
C04378=1175.190,227.561,-62.799,-177.572,7.110,148.620
C04379=1175.195,227.313,-62.774,-177.575,7.107,148.621
C04380=1175.199,227.064,-62.748,-177.577,7.105,148.621
C04381=1175.204,226.816,-62.723,-177.581,7.102,148.621
C04382=1175.208,226.568,-62.697,-177.583,7.100,148.621
C04383=1175.213,226.318,-62.672,-177.586,7.098,148.621
C04384=1175.217,226.069,-62.646,-177.588,7.096,148.622
C04385=1175.222,225.821,-62.621,-177.591,7.093,148.622
C04386=1175.226,225.572,-62.595,-177.594,7.091,148.622
C04387=1175.230,225.324,-62.570,-177.597,7.088,148.622
C04388=1175.235,225.076,-62.544,-177.599,7.086,148.622
C04389=1175.240,224.826,-62.519,-177.602,7.083,148.623
C04390=1175.244,224.577,-62.493,-177.604,7.081,148.623
C04391=1175.249,224.329,-62.468,-177.607,7.079,148.623
C04392=1175.253,224.080,-62.442,-177.610,7.076,148.623
C04393=1175.258,223.832,-62.418,-177.612,7.075,148.623
C04394=1175.262,223.583,-62.392,-177.615,7.072,148.624
C04395=1175.266,223.334,-62.367,-177.618,7.070,148.624
C04396=1175.271,223.086,-62.342,-177.621,7.067,148.624
C04397=1175.275,222.837,-62.316,-177.623,7.065,148.624
C04398=1175.280,222.589,-62.291,-177.626,7.063,148.625
C04399=1175.285,222.339,-62.266,-177.629,7.060,148.625
C04400=1175.289,222.091,-62.240,-177.631,7.059,148.625
C04401=1175.294,221.842,-62.215,-177.634,7.056,148.625
C04402=1175.298,221.593,-62.190,-177.637,7.054,148.625
C04403=1175.303,221.345,-62.164,-177.639,7.051,148.626
C04404=1175.307,221.096,-62.139,-177.642,7.049,148.626
C04405=1175.312,220.848,-62.114,-177.644,7.047,148.626
C04406=1175.316,220.599,-62.089,-177.648,7.044,148.626
C04407=1175.321,220.350,-62.064,-177.650,7.042,148.626
C04408=1175.325,220.101,-62.038,-177.653,7.040,148.627
C04409=1175.330,219.853,-62.014,-177.655,7.037,148.627
C04410=1175.334,219.604,-61.988,-177.658,7.035,148.627
C04411=1175.339,219.355,-61.964,-177.661,7.033,148.627
C04412=1175.343,219.107,-61.938,-177.663,7.031,148.628
C04413=1175.348,218.858,-61.913,-177.666,7.028,148.628
C04414=1175.352,218.609,-61.888,-177.669,7.026,148.628
C04415=1175.357,218.361,-61.864,-177.672,7.024,148.628
C04416=1175.361,218.112,-61.838,-177.674,7.021,148.628
C04417=1175.366,217.863,-61.813,-177.677,7.020,148.629
C04418=1175.370,217.615,-61.788,-177.680,7.017,148.629
C04419=1175.375,217.366,-61.763,-177.682,7.015,148.629
C04420=1175.379,217.117,-61.738,-177.685,7.012,148.630
C04421=1175.384,216.869,-61.713,-177.688,7.010,148.630
C04422=1175.388,216.619,-61.688,-177.690,7.008,148.630
C04423=1175.393,216.371,-61.663,-177.693,7.005,148.630
C04424=1175.397,216.122,-61.638,-177.696,7.004,148.630
C04425=1175.402,215.873,-61.614,-177.699,7.001,148.631
C04426=1175.407,215.625,-61.589,-177.701,6.999,148.631
C04427=1175.411,215.376,-61.564,-177.704,6.997,148.631
C04428=1175.416,215.127,-61.539,-177.706,6.994,148.631
C04429=1175.420,214.879,-61.514,-177.709,6.992,148.632
C04430=1175.424,214.630,-61.490,-177.712,6.990,148.632
C04431=1175.429,214.381,-61.465,-177.715,6.988,148.632
C04432=1175.434,214.132,-61.440,-177.717,6.986,148.632
C04433=1175.438,213.884,-61.415,-177.720,6.983,148.632
C04434=1175.442,213.635,-61.390,-177.723,6.981,148.633
C04435=1175.448,213.386,-61.365,-177.725,6.979,148.633
C04436=1175.451,213.137,-61.341,-177.728,6.976,148.633
C04437=1175.456,212.889,-61.316,-177.731,6.974,148.634
C04438=1175.461,212.640,-61.292,-177.733,6.972,148.634
C04439=1175.465,212.391,-61.266,-177.736,6.970,148.634
C04440=1175.470,212.143,-61.242,-177.739,6.968,148.634
C04441=1175.475,211.894,-61.218,-177.742,6.965,148.634
C04442=1175.478,211.645,-61.193,-177.744,6.963,148.635
C04443=1175.483,211.397,-61.168,-177.746,6.961,148.635
C04444=1175.488,211.148,-61.143,-177.750,6.958,148.635
C04445=1175.492,210.899,-61.119,-177.752,6.957,148.636
C04446=1175.497,210.629,-61.092,-177.756,6.954,148.636
C04447=1175.503,210.358,-61.066,-177.758,6.952,148.636
C04448=1175.507,210.087,-61.039,-177.761,6.949,148.636
C04449=1175.513,209.817,-61.012,-177.764,6.947,148.637
C04450=1175.517,209.568,-60.988,-177.766,6.945,148.637
C04451=1175.521,209.319,-60.963,-177.769,6.943,148.637
C04452=1175.526,209.071,-60.939,-177.772,6.940,148.637
C04453=1175.531,208.822,-60.914,-177.775,6.938,148.637
C04454=1175.535,208.573,-60.890,-177.777,6.936,148.638
C04455=1175.540,208.324,-60.865,-177.780,6.934,148.638
C04456=1175.544,208.076,-60.841,-177.783,6.931,148.638
C04457=1175.549,207.827,-60.817,-177.785,6.930,148.639
C04458=1175.553,207.578,-60.792,-177.789,6.927,148.639
C04459=1175.558,207.329,-60.768,-177.791,6.925,148.639
C04460=1175.563,207.081,-60.743,-177.793,6.923,148.639
C04461=1175.567,206.832,-60.719,-177.797,6.921,148.640
C04462=1175.571,206.583,-60.695,-177.799,6.918,148.640
C04463=1175.576,206.334,-60.670,-177.801,6.917,148.640
C04464=1175.580,206.086,-60.646,-177.805,6.914,148.640
C04465=1175.585,205.837,-60.623,-177.807,6.912,148.641
C04466=1175.590,205.587,-60.598,-177.810,6.910,148.641
C04467=1175.594,205.339,-60.574,-177.812,6.908,148.641
C04468=1175.599,205.090,-60.549,-177.815,6.905,148.641
C04469=1175.604,204.842,-60.525,-177.818,6.904,148.642
C04470=1175.607,204.593,-60.501,-177.820,6.902,148.642
C04471=1175.612,204.344,-60.477,-177.823,6.899,148.642
C04472=1175.617,204.095,-60.452,-177.826,6.897,148.642
C04473=1175.622,203.847,-60.428,-177.828,6.895,148.643
C04474=1175.626,203.598,-60.404,-177.831,6.892,148.643
C04475=1175.631,203.348,-60.380,-177.834,6.891,148.643
C04476=1175.635,203.100,-60.356,-177.837,6.889,148.644
C04477=1175.640,202.851,-60.332,-177.839,6.887,148.644
C04478=1175.644,202.603,-60.308,-177.842,6.884,148.644
C04479=1175.650,202.354,-60.284,-177.845,6.882,148.644
C04480=1175.653,202.105,-60.259,-177.847,6.880,148.645
C04481=1175.658,201.856,-60.235,-177.850,6.877,148.645
C04482=1175.662,201.607,-60.212,-177.853,6.876,148.645
C04483=1175.668,201.358,-60.187,-177.855,6.874,148.646
C04484=1175.672,201.110,-60.163,-177.858,6.871,148.646
C04485=1175.677,200.861,-60.140,-177.861,6.869,148.646
C04486=1175.681,200.612,-60.116,-177.863,6.867,148.646
C04487=1175.685,200.363,-60.092,-177.866,6.865,148.646
C04488=1175.690,200.114,-60.068,-177.869,6.863,148.647
C04489=1175.695,199.866,-60.043,-177.872,6.861,148.647
C04490=1175.699,199.617,-60.020,-177.874,6.859,148.647
C04491=1175.704,199.368,-59.996,-177.876,6.857,148.648
C04492=1175.708,199.119,-59.973,-177.880,6.854,148.648
C04493=1175.713,198.871,-59.948,-177.882,6.853,148.648
C04494=1175.718,198.622,-59.925,-177.885,6.850,148.648
C04495=1175.722,198.373,-59.901,-177.888,6.848,148.649
C04496=1175.727,198.123,-59.877,-177.890,6.846,148.649
C04497=1175.731,197.875,-59.853,-177.893,6.844,148.649
C04498=1175.736,197.626,-59.829,-177.895,6.842,148.650
C04499=1175.740,197.377,-59.805,-177.899,6.840,148.650
C04500=1175.745,197.128,-59.782,-177.901,6.838,148.650
C04501=1175.749,196.880,-59.758,-177.904,6.836,148.651
C04502=1175.754,196.631,-59.734,-177.906,6.834,148.651
C04503=1175.759,196.382,-59.711,-177.909,6.831,148.651
C04504=1175.763,196.133,-59.687,-177.912,6.829,148.651
C04505=1175.768,195.884,-59.664,-177.914,6.827,148.652
C04506=1175.772,195.636,-59.640,-177.917,6.826,148.652
C04507=1175.777,195.387,-59.616,-177.920,6.823,148.652
C04508=1175.782,195.138,-59.593,-177.923,6.821,148.653
C04509=1175.786,194.890,-59.569,-177.925,6.819,148.653
C04510=1175.791,194.641,-59.545,-177.928,6.817,148.653
C04511=1175.795,194.391,-59.522,-177.931,6.815,148.653
C04512=1175.800,194.143,-59.498,-177.934,6.813,148.654
C04513=1175.805,193.894,-59.475,-177.936,6.811,148.654
C04514=1175.809,193.645,-59.451,-177.938,6.809,148.654
C04515=1175.814,193.397,-59.427,-177.941,6.807,148.655
C04516=1175.818,193.148,-59.404,-177.944,6.805,148.655
C04517=1175.823,192.899,-59.380,-177.947,6.803,148.655
C04518=1175.828,192.649,-59.357,-177.949,6.801,148.655
C04519=1175.832,192.401,-59.333,-177.952,6.799,148.656
C04520=1175.837,192.152,-59.310,-177.955,6.796,148.656
C04521=1175.841,191.903,-59.286,-177.958,6.795,148.656
C04522=1175.846,191.654,-59.263,-177.960,6.792,148.656
C04523=1175.851,191.405,-59.240,-177.963,6.791,148.657
C04524=1175.856,191.156,-59.216,-177.965,6.789,148.657
C04525=1175.860,190.907,-59.192,-177.969,6.786,148.658
C04526=1175.864,190.659,-59.169,-177.971,6.784,148.658
C04527=1175.869,190.410,-59.146,-177.973,6.782,148.658
C04528=1175.873,190.161,-59.123,-177.976,6.781,148.658
C04529=1175.878,189.912,-59.099,-177.979,6.779,148.659
C04530=1175.883,189.663,-59.076,-177.982,6.776,148.659
C04531=1175.887,189.414,-59.053,-177.985,6.774,148.659
C04532=1175.893,189.165,-59.030,-177.987,6.772,148.660
C04533=1175.897,188.917,-59.007,-177.990,6.771,148.660
C04534=1175.901,188.668,-58.983,-177.992,6.769,148.660
C04535=1175.906,188.419,-58.959,-177.996,6.766,148.661
C04536=1175.911,188.170,-58.936,-177.998,6.764,148.661
C04537=1175.915,187.921,-58.913,-178.000,6.762,148.661
C04538=1175.919,187.672,-58.890,-178.003,6.760,148.661
C04539=1175.924,187.423,-58.867,-178.006,6.759,148.662
C04540=1175.929,187.174,-58.843,-178.009,6.756,148.662
C04541=1175.934,186.926,-58.820,-178.012,6.754,148.662
C04542=1175.939,186.677,-58.797,-178.014,6.752,148.663
C04543=1175.943,186.428,-58.774,-178.017,6.750,148.663
C04544=1175.948,186.179,-58.751,-178.019,6.749,148.663
C04545=1175.952,185.929,-58.728,-178.022,6.746,148.664
C04546=1175.956,185.681,-58.705,-178.025,6.744,148.664
C04547=1175.961,185.432,-58.682,-178.027,6.742,148.664
C04548=1175.966,185.183,-58.659,-178.030,6.740,148.664
C04549=1175.971,184.934,-58.636,-178.033,6.739,148.665
C04550=1175.975,184.665,-58.611,-178.036,6.736,148.665
C04551=1175.981,184.395,-58.586,-178.039,6.734,148.666
C04552=1175.986,184.125,-58.561,-178.041,6.732,148.666
C04553=1175.991,183.856,-58.537,-178.045,6.730,148.666
C04554=1175.995,183.607,-58.513,-178.047,6.728,148.667
C04555=1175.999,183.358,-58.491,-178.050,6.726,148.667
C04556=1176.004,183.109,-58.467,-178.053,6.724,148.667
C04557=1176.009,182.860,-58.444,-178.055,6.722,148.667
C04558=1176.014,182.611,-58.422,-178.058,6.720,148.668
C04559=1176.018,182.362,-58.399,-178.061,6.718,148.668
C04560=1176.023,182.113,-58.375,-178.063,6.716,148.668
C04561=1176.027,181.865,-58.353,-178.066,6.714,148.669
C04562=1176.033,181.616,-58.330,-178.069,6.713,148.669
C04563=1176.037,181.367,-58.308,-178.071,6.711,148.670
C04564=1176.041,181.118,-58.284,-178.074,6.708,148.670
C04565=1176.046,180.869,-58.261,-178.077,6.706,148.670
C04566=1176.051,180.620,-58.239,-178.080,6.704,148.670
C04567=1176.056,180.371,-58.216,-178.082,6.703,148.671
C04568=1176.059,180.123,-58.193,-178.085,6.701,148.671
C04569=1176.065,179.873,-58.170,-178.088,6.699,148.671
C04570=1176.069,179.625,-58.148,-178.090,6.697,148.672
C04571=1176.074,179.376,-58.125,-178.093,6.694,148.672
C04572=1176.078,179.127,-58.103,-178.096,6.693,148.672
C04573=1176.083,178.877,-58.079,-178.098,6.691,148.673
C04574=1176.088,178.629,-58.058,-178.101,6.689,148.673
C04575=1176.092,178.380,-58.034,-178.104,6.687,148.673
C04576=1176.097,178.130,-58.012,-178.106,6.686,148.674
C04577=1176.102,177.882,-57.989,-178.109,6.684,148.674
C04578=1176.106,177.633,-57.966,-178.112,6.682,148.674
C04579=1176.111,177.384,-57.944,-178.114,6.680,148.675
C04580=1176.115,177.136,-57.921,-178.117,6.677,148.675
C04581=1176.120,176.886,-57.899,-178.120,6.675,148.675
C04582=1176.124,176.637,-57.876,-178.123,6.674,148.676
C04583=1176.130,176.388,-57.854,-178.125,6.672,148.676
C04584=1176.134,176.140,-57.831,-178.128,6.670,148.676
C04585=1176.138,175.890,-57.809,-178.131,6.668,148.677
C04586=1176.144,175.642,-57.786,-178.133,6.667,148.677
C04587=1176.148,175.393,-57.764,-178.136,6.665,148.678
C04588=1176.153,175.143,-57.741,-178.138,6.663,148.678
C04589=1176.157,174.895,-57.719,-178.141,6.660,148.678
C04590=1176.162,174.646,-57.697,-178.144,6.658,148.678
C04591=1176.166,174.397,-57.673,-178.147,6.657,148.679
C04592=1176.171,174.148,-57.652,-178.149,6.655,148.679
C04593=1176.176,173.898,-57.629,-178.152,6.653,148.679
C04594=1176.181,173.650,-57.607,-178.155,6.651,148.680
C04595=1176.185,173.401,-57.585,-178.157,6.650,148.680
C04596=1176.190,173.152,-57.561,-178.160,6.648,148.681
C04597=1176.195,172.903,-57.540,-178.163,6.646,148.681
C04598=1176.199,172.654,-57.518,-178.166,6.644,148.681
C04599=1176.204,172.405,-57.495,-178.168,6.642,148.682
C04600=1176.208,172.156,-57.472,-178.171,6.640,148.682
C04601=1176.213,171.907,-57.450,-178.174,6.638,148.682
C04602=1176.218,171.658,-57.429,-178.176,6.636,148.682
C04603=1176.222,171.409,-57.405,-178.179,6.634,148.683
C04604=1176.227,171.161,-57.384,-178.182,6.632,148.683
C04605=1176.231,170.911,-57.362,-178.184,6.631,148.684
C04606=1176.237,170.662,-57.339,-178.187,6.629,148.684
C04607=1176.241,170.414,-57.317,-178.190,6.627,148.684
C04608=1176.245,170.164,-57.295,-178.192,6.625,148.685
C04609=1176.250,169.916,-57.273,-178.195,6.624,148.685
C04610=1176.255,169.666,-57.250,-178.198,6.622,148.685
C04611=1176.260,169.417,-57.229,-178.200,6.620,148.686
C04612=1176.264,169.168,-57.207,-178.203,6.618,148.686
C04613=1176.269,168.920,-57.184,-178.206,6.617,148.687
C04614=1176.273,168.671,-57.162,-178.209,6.615,148.687
C04615=1176.279,168.422,-57.140,-178.211,6.612,148.687
C04616=1176.283,168.172,-57.118,-178.214,6.610,148.687
C04617=1176.288,167.924,-57.096,-178.217,6.608,148.688
C04618=1176.292,167.674,-57.074,-178.219,6.607,148.688
C04619=1176.297,167.426,-57.052,-178.222,6.605,148.688
C04620=1176.302,167.176,-57.030,-178.225,6.603,148.689
C04621=1176.307,166.927,-57.008,-178.227,6.601,148.689
C04622=1176.311,166.678,-56.986,-178.230,6.599,148.690
C04623=1176.316,166.430,-56.964,-178.233,6.598,148.690
C04624=1176.320,166.181,-56.942,-178.235,6.596,148.690
C04625=1176.325,165.932,-56.920,-178.238,6.594,148.691
C04626=1176.329,165.683,-56.898,-178.241,6.592,148.691
C04627=1176.334,165.434,-56.876,-178.244,6.591,148.691
C04628=1176.340,165.185,-56.854,-178.246,6.589,148.692
C04629=1176.344,164.936,-56.832,-178.249,6.587,148.692
C04630=1176.349,164.687,-56.810,-178.252,6.585,148.693
C04631=1176.353,164.437,-56.789,-178.254,6.584,148.693
C04632=1176.358,164.189,-56.767,-178.257,6.582,148.693
C04633=1176.362,163.939,-56.745,-178.260,6.580,148.694
C04634=1176.367,163.691,-56.723,-178.262,6.578,148.694
C04635=1176.372,163.442,-56.702,-178.265,6.577,148.694
C04636=1176.376,163.193,-56.680,-178.268,6.575,148.695
C04637=1176.381,162.944,-56.658,-178.270,6.573,148.695
C04638=1176.386,162.695,-56.636,-178.273,6.571,148.696
C04639=1176.390,162.446,-56.614,-178.276,6.569,148.696
C04640=1176.395,162.197,-56.592,-178.278,6.568,148.696
C04641=1176.400,161.947,-56.571,-178.281,6.566,148.697
C04642=1176.405,161.699,-56.550,-178.284,6.564,148.697
C04643=1176.409,161.449,-56.527,-178.286,6.562,148.697
C04644=1176.414,161.201,-56.506,-178.289,6.561,148.698
C04645=1176.419,160.952,-56.484,-178.292,6.559,148.698
C04646=1176.423,160.702,-56.463,-178.295,6.557,148.698
C04647=1176.428,160.454,-56.441,-178.297,6.555,148.699
C04648=1176.432,160.204,-56.419,-178.300,6.554,148.699
C04649=1176.437,159.956,-56.397,-178.303,6.552,148.700
C04650=1176.442,159.706,-56.376,-178.305,6.550,148.700
C04651=1176.447,159.457,-56.354,-178.308,6.548,148.700
C04652=1176.452,159.208,-56.333,-178.311,6.547,148.701
C04653=1176.456,158.960,-56.311,-178.313,6.545,148.701
C04654=1176.461,158.691,-56.288,-178.316,6.543,148.701
C04655=1176.467,158.421,-56.265,-178.319,6.540,148.702
C04656=1176.471,158.152,-56.242,-178.322,6.539,148.702
C04657=1176.477,157.883,-56.218,-178.325,6.537,148.703
C04658=1176.481,157.635,-56.198,-178.328,6.536,148.703
C04659=1176.485,157.385,-56.176,-178.331,6.534,148.704
C04660=1176.490,157.137,-56.154,-178.333,6.532,148.704
C04661=1176.495,156.887,-56.133,-178.336,6.530,148.704
C04662=1176.500,156.639,-56.111,-178.339,6.528,148.705
C04663=1176.505,156.389,-56.090,-178.341,6.527,148.705
C04664=1176.509,156.140,-56.069,-178.344,6.525,148.705
C04665=1176.514,155.892,-56.047,-178.347,6.523,148.706
C04666=1176.519,155.642,-56.026,-178.349,6.521,148.706
C04667=1176.523,155.393,-56.004,-178.352,6.520,148.707
C04668=1176.528,155.144,-55.983,-178.355,6.518,148.707
C04669=1176.533,154.895,-55.961,-178.357,6.516,148.707
C04670=1176.537,154.646,-55.941,-178.360,6.514,148.708
C04671=1176.542,154.397,-55.919,-178.363,6.513,148.708
C04672=1176.547,154.148,-55.898,-178.365,6.511,148.708
C04673=1176.552,153.899,-55.876,-178.368,6.509,148.709
C04674=1176.557,153.650,-55.856,-178.370,6.508,148.709
C04675=1176.561,153.401,-55.834,-178.373,6.506,148.710
C04676=1176.566,153.151,-55.813,-178.376,6.505,148.710
C04677=1176.571,152.903,-55.791,-178.378,6.503,148.710
C04678=1176.575,152.654,-55.771,-178.381,6.501,148.711
C04679=1176.580,152.404,-55.750,-178.384,6.500,148.711
C04680=1176.585,152.155,-55.728,-178.387,6.498,148.712
C04681=1176.589,151.906,-55.708,-178.390,6.496,148.712
C04682=1176.594,151.658,-55.686,-178.392,6.495,148.712
C04683=1176.599,151.408,-55.665,-178.395,6.493,148.713
C04684=1176.604,151.159,-55.644,-178.398,6.491,148.713
C04685=1176.608,150.910,-55.623,-178.400,6.489,148.714
C04686=1176.613,150.661,-55.602,-178.403,6.487,148.714
C04687=1176.618,150.412,-55.581,-178.406,6.486,148.714
C04688=1176.622,150.163,-55.559,-178.408,6.484,148.715
C04689=1176.628,149.914,-55.539,-178.411,6.482,148.715
C04690=1176.633,149.665,-55.518,-178.413,6.481,148.716
C04691=1176.636,149.416,-55.496,-178.416,6.480,148.716
C04692=1176.641,149.166,-55.475,-178.419,6.478,148.716
C04693=1176.646,148.918,-55.455,-178.422,6.476,148.717
C04694=1176.651,148.668,-55.434,-178.425,6.475,148.717
C04695=1176.656,148.420,-55.412,-178.427,6.473,148.718
C04696=1176.660,148.171,-55.392,-178.430,6.471,148.718
C04697=1176.666,147.921,-55.371,-178.433,6.469,148.718
C04698=1176.669,147.672,-55.350,-178.435,6.468,148.719
C04699=1176.674,147.423,-55.328,-178.438,6.466,148.719
C04700=1176.679,147.174,-55.308,-178.441,6.464,148.720
C04701=1176.684,146.925,-55.287,-178.443,6.463,148.720
C04702=1176.689,146.676,-55.266,-178.445,6.461,148.720
C04703=1176.693,146.427,-55.246,-178.448,6.460,148.721
C04704=1176.699,146.177,-55.225,-178.451,6.458,148.721
C04705=1176.703,145.929,-55.204,-178.454,6.456,148.722
C04706=1176.708,145.680,-55.183,-178.457,6.455,148.722
C04707=1176.712,145.431,-55.162,-178.459,6.453,148.722
C04708=1176.718,145.182,-55.141,-178.462,6.451,148.723
C04709=1176.721,144.932,-55.121,-178.465,6.449,148.723
C04710=1176.727,144.683,-55.100,-178.467,6.448,148.724
C04711=1176.731,144.434,-55.079,-178.470,6.447,148.724
C04712=1176.736,144.185,-55.058,-178.472,6.445,148.724
C04713=1176.741,143.936,-55.038,-178.475,6.444,148.725
C04714=1176.746,143.686,-55.017,-178.478,6.442,148.725
C04715=1176.750,143.437,-54.997,-178.481,6.440,148.726
C04716=1176.755,143.188,-54.976,-178.484,6.438,148.726
C04717=1176.760,142.939,-54.955,-178.486,6.437,148.727
C04718=1176.764,142.690,-54.935,-178.489,6.435,148.727
C04719=1176.769,142.441,-54.914,-178.491,6.434,148.727
C04720=1176.774,142.192,-54.894,-178.494,6.432,148.728
C04721=1176.779,141.943,-54.873,-178.497,6.431,148.728
C04722=1176.783,141.694,-54.852,-178.500,6.429,148.729
C04723=1176.788,141.445,-54.832,-178.502,6.427,148.729
C04724=1176.793,141.196,-54.811,-178.505,6.426,148.729
C04725=1176.798,140.947,-54.790,-178.508,6.424,148.730
C04726=1176.802,140.698,-54.770,-178.510,6.423,148.730
C04727=1176.807,140.448,-54.749,-178.513,6.421,148.731
C04728=1176.812,140.200,-54.729,-178.516,6.420,148.731
C04729=1176.817,139.950,-54.708,-178.518,6.418,148.732
C04730=1176.821,139.701,-54.687,-178.521,6.416,148.732
C04731=1176.826,139.452,-54.668,-178.524,6.414,148.732
C04732=1176.831,139.202,-54.647,-178.527,6.413,148.733
C04733=1176.836,138.954,-54.626,-178.529,6.412,148.733
C04734=1176.840,138.705,-54.606,-178.531,6.410,148.734
C04735=1176.844,138.456,-54.586,-178.535,6.409,148.734
C04736=1176.850,138.206,-54.565,-178.537,6.407,148.735
C04737=1176.854,137.957,-54.545,-178.540,6.405,148.735
C04738=1176.859,137.708,-54.525,-178.543,6.403,148.735
C04739=1176.864,137.459,-54.504,-178.545,6.402,148.736
C04740=1176.869,137.210,-54.484,-178.547,6.401,148.736
C04741=1176.874,136.961,-54.464,-178.551,6.399,148.737
C04742=1176.878,136.712,-54.444,-178.553,6.398,148.737
C04743=1176.883,136.463,-54.423,-178.556,6.396,148.738
C04744=1176.888,136.214,-54.402,-178.559,6.394,148.738
C04745=1176.893,135.964,-54.383,-178.561,6.393,148.738
C04746=1176.897,135.715,-54.362,-178.564,6.391,148.739
C04747=1176.902,135.466,-54.341,-178.567,6.390,148.739
C04748=1176.907,135.216,-54.322,-178.569,6.388,148.740
C04749=1176.911,134.967,-54.301,-178.572,6.387,148.740
C04750=1176.916,134.719,-54.281,-178.575,6.385,148.740
C04751=1176.921,134.470,-54.262,-178.577,6.384,148.741
C04752=1176.926,134.220,-54.241,-178.580,6.382,148.741
C04753=1176.931,133.971,-54.220,-178.583,6.381,148.742
C04754=1176.935,133.722,-54.201,-178.585,6.379,148.742
C04755=1176.940,133.473,-54.180,-178.588,6.377,148.743
C04756=1176.945,133.223,-54.161,-178.590,6.376,148.743
C04757=1176.950,132.975,-54.141,-178.593,6.375,148.743
C04758=1176.955,132.706,-54.119,-178.596,6.373,148.744
C04759=1176.960,132.438,-54.097,-178.599,6.371,148.744
C04760=1176.966,132.169,-54.075,-178.602,6.370,148.745
C04761=1176.970,131.900,-54.054,-178.605,6.368,148.745
C04762=1176.975,131.651,-54.034,-178.607,6.367,148.746
C04763=1176.980,131.402,-54.013,-178.610,6.365,148.746
C04764=1176.985,131.153,-53.993,-178.613,6.363,148.747
C04765=1176.989,130.904,-53.973,-178.616,6.362,148.747
C04766=1176.994,130.654,-53.953,-178.618,6.361,148.748
C04767=1176.999,130.405,-53.934,-178.621,6.359,148.748
C04768=1177.004,130.156,-53.914,-178.624,6.357,148.748
C04769=1177.009,129.907,-53.894,-178.626,6.356,148.749
C04770=1177.013,129.658,-53.874,-178.629,6.355,148.749
C04771=1177.018,129.409,-53.854,-178.632,6.353,148.750
C04772=1177.023,129.160,-53.834,-178.634,6.351,148.750
C04773=1177.028,128.910,-53.814,-178.637,6.350,148.751
C04774=1177.032,128.661,-53.795,-178.640,6.348,148.751
C04775=1177.037,128.412,-53.774,-178.642,6.347,148.752
C04776=1177.042,128.163,-53.755,-178.645,6.346,148.752
C04777=1177.046,127.914,-53.735,-178.648,6.344,148.752
C04778=1177.051,127.664,-53.715,-178.650,6.342,148.753
C04779=1177.056,127.415,-53.695,-178.653,6.341,148.753
C04780=1177.061,127.167,-53.675,-178.656,6.340,148.754
C04781=1177.066,126.917,-53.656,-178.658,6.338,148.754
C04782=1177.070,126.667,-53.636,-178.661,6.336,148.755
C04783=1177.076,126.419,-53.616,-178.663,6.335,148.755
C04784=1177.080,126.170,-53.596,-178.666,6.334,148.756
C04785=1177.085,125.920,-53.577,-178.669,6.332,148.756
C04786=1177.089,125.671,-53.556,-178.672,6.331,148.756
C04787=1177.095,125.422,-53.537,-178.675,6.329,148.757
C04788=1177.100,125.173,-53.517,-178.677,6.328,148.758
C04789=1177.104,124.923,-53.498,-178.680,6.327,148.758
C04790=1177.109,124.675,-53.478,-178.683,6.325,148.758
C04791=1177.114,124.425,-53.458,-178.685,6.323,148.759
C04792=1177.118,124.176,-53.439,-178.688,6.323,148.759
C04793=1177.123,123.927,-53.419,-178.691,6.321,148.760
C04794=1177.128,123.678,-53.400,-178.693,6.319,148.760
C04795=1177.133,123.429,-53.380,-178.695,6.318,148.761
C04796=1177.137,123.179,-53.360,-178.698,6.316,148.761
C04797=1177.143,122.930,-53.341,-178.701,6.315,148.762
C04798=1177.147,122.681,-53.321,-178.704,6.313,148.762
C04799=1177.151,122.431,-53.302,-178.706,6.312,148.762
C04800=1177.157,122.183,-53.283,-178.709,6.311,148.763
C04801=1177.162,121.933,-53.263,-178.712,6.309,148.763
C04802=1177.167,121.685,-53.243,-178.715,6.307,148.764
C04803=1177.171,121.435,-53.223,-178.717,6.307,148.764
C04804=1177.176,121.186,-53.204,-178.720,6.305,148.765
C04805=1177.181,120.937,-53.185,-178.723,6.303,148.765
C04806=1177.185,120.688,-53.165,-178.725,6.302,148.766
C04807=1177.190,120.438,-53.146,-178.728,6.301,148.766
C04808=1177.195,120.189,-53.126,-178.731,6.299,148.767
C04809=1177.200,119.939,-53.107,-178.733,6.298,148.767
C04810=1177.205,119.691,-53.088,-178.736,6.297,148.767
C04811=1177.210,119.441,-53.068,-178.738,6.295,148.768
C04812=1177.214,119.192,-53.049,-178.741,6.294,148.768
C04813=1177.220,118.943,-53.030,-178.744,6.292,148.769
C04814=1177.224,118.694,-53.010,-178.746,6.291,148.769
C04815=1177.229,118.445,-52.991,-178.749,6.289,148.770
C04816=1177.234,118.195,-52.972,-178.752,6.288,148.770
C04817=1177.239,117.946,-52.952,-178.754,6.287,148.771
C04818=1177.243,117.697,-52.933,-178.757,6.285,148.771
C04819=1177.248,117.448,-52.914,-178.760,6.284,148.772
C04820=1177.253,117.199,-52.894,-178.762,6.283,148.772
C04821=1177.257,116.949,-52.875,-178.765,6.281,148.773
C04822=1177.263,116.701,-52.856,-178.768,6.279,148.773
C04823=1177.268,116.450,-52.837,-178.771,6.278,148.774
C04824=1177.272,116.202,-52.818,-178.773,6.277,148.774
C04825=1177.277,115.952,-52.799,-178.776,6.275,148.774
C04826=1177.282,115.703,-52.779,-178.779,6.274,148.775
C04827=1177.286,115.454,-52.760,-178.781,6.273,148.775
C04828=1177.292,115.205,-52.741,-178.784,6.271,148.776
C04829=1177.296,114.956,-52.721,-178.787,6.270,148.776
C04830=1177.301,114.707,-52.703,-178.789,6.269,148.777
C04831=1177.306,114.457,-52.684,-178.792,6.267,148.777
C04832=1177.311,114.208,-52.664,-178.795,6.266,148.778
C04833=1177.315,113.959,-52.645,-178.797,6.265,148.778
C04834=1177.321,113.710,-52.626,-178.800,6.263,148.779
C04835=1177.325,113.460,-52.608,-178.803,6.262,148.779
C04836=1177.330,113.211,-52.588,-178.805,6.261,148.780
C04837=1177.335,112.962,-52.569,-178.808,6.259,148.780
C04838=1177.340,112.713,-52.550,-178.811,6.258,148.781
C04839=1177.345,112.463,-52.531,-178.813,6.257,148.781
C04840=1177.349,112.214,-52.512,-178.816,6.255,148.782
C04841=1177.354,111.965,-52.493,-178.819,6.254,148.782
C04842=1177.359,111.716,-52.475,-178.821,6.253,148.782
C04843=1177.364,111.466,-52.455,-178.824,6.251,148.783
C04844=1177.368,111.217,-52.436,-178.827,6.250,148.783
C04845=1177.373,110.967,-52.417,-178.829,6.249,148.784
C04846=1177.378,110.719,-52.399,-178.832,6.247,148.785
C04847=1177.383,110.470,-52.379,-178.835,6.246,148.785
C04848=1177.388,110.220,-52.361,-178.837,6.245,148.785
C04849=1177.393,109.971,-52.342,-178.840,6.243,148.786
C04850=1177.397,109.722,-52.323,-178.843,6.242,148.786
C04851=1177.403,109.472,-52.304,-178.845,6.241,148.787
C04852=1177.407,109.223,-52.285,-178.848,6.239,148.787
C04853=1177.412,108.974,-52.267,-178.851,6.238,148.788
C04854=1177.417,108.725,-52.248,-178.853,6.237,148.788
C04855=1177.422,108.476,-52.228,-178.856,6.235,148.789
C04856=1177.427,108.226,-52.210,-178.859,6.234,148.789
C04857=1177.431,107.977,-52.191,-178.861,6.233,148.790
C04858=1177.436,107.728,-52.173,-178.864,6.231,148.790
C04859=1177.442,107.479,-52.153,-178.866,6.230,148.791
C04860=1177.446,107.229,-52.135,-178.869,6.229,148.791
C04861=1177.451,106.980,-52.116,-178.872,6.227,148.792
C04862=1177.456,106.712,-52.096,-178.875,6.226,148.792
C04863=1177.461,106.443,-52.076,-178.878,6.225,148.793
C04864=1177.466,106.175,-52.056,-178.880,6.223,148.793
C04865=1177.472,105.906,-52.036,-178.883,6.222,148.794
C04866=1177.476,105.657,-52.017,-178.886,6.220,148.794
C04867=1177.481,105.408,-51.999,-178.888,6.219,148.795
C04868=1177.486,105.159,-51.979,-178.891,6.218,148.795
C04869=1177.491,104.909,-51.961,-178.894,6.217,148.796
C04870=1177.496,104.660,-51.943,-178.896,6.215,148.796
C04871=1177.501,104.411,-51.924,-178.900,6.214,148.797
C04872=1177.505,104.161,-51.905,-178.902,6.213,148.797
C04873=1177.510,103.913,-51.887,-178.904,6.211,148.798
C04874=1177.516,103.663,-51.868,-178.908,6.210,148.798
C04875=1177.520,103.414,-51.850,-178.910,6.209,148.799
C04876=1177.524,103.165,-51.831,-178.912,6.207,148.799
C04877=1177.530,102.915,-51.813,-178.915,6.207,148.800
C04878=1177.535,102.666,-51.795,-178.918,6.205,148.800
C04879=1177.539,102.417,-51.776,-178.921,6.204,148.801
C04880=1177.545,102.167,-51.757,-178.923,6.203,148.801
C04881=1177.550,101.918,-51.739,-178.926,6.201,148.802
C04882=1177.554,101.669,-51.720,-178.928,6.200,148.802
C04883=1177.559,101.420,-51.702,-178.931,6.199,148.803
C04884=1177.564,101.170,-51.683,-178.934,6.197,148.803
C04885=1177.569,100.921,-51.665,-178.936,6.196,148.804
C04886=1177.573,100.672,-51.646,-178.939,6.195,148.804
C04887=1177.578,100.423,-51.628,-178.941,6.194,148.805
C04888=1177.584,100.173,-51.610,-178.945,6.192,148.805
C04889=1177.589,99.924,-51.592,-178.947,6.191,148.806
C04890=1177.593,99.675,-51.573,-178.950,6.190,148.806
C04891=1177.597,99.425,-51.555,-178.953,6.188,148.807
C04892=1177.602,99.176,-51.537,-178.955,6.188,148.807
C04893=1177.608,98.927,-51.518,-178.958,6.186,148.808
C04894=1177.612,98.677,-51.500,-178.960,6.185,148.808
C04895=1177.617,98.428,-51.481,-178.963,6.184,148.809
C04896=1177.622,98.179,-51.463,-178.966,6.182,148.809
C04897=1177.627,97.930,-51.445,-178.968,6.181,148.810
C04898=1177.632,97.681,-51.427,-178.971,6.180,148.810
C04899=1177.637,97.431,-51.408,-178.973,6.179,148.811
C04900=1177.642,97.181,-51.390,-178.976,6.177,148.811
C04901=1177.647,96.932,-51.372,-178.979,6.177,148.812
C04902=1177.651,96.683,-51.354,-178.981,6.175,148.812
C04903=1177.656,96.435,-51.336,-178.984,6.174,148.813
C04904=1177.660,96.185,-51.317,-178.987,6.173,148.813
C04905=1177.665,95.936,-51.299,-178.990,6.171,148.814
C04906=1177.670,95.686,-51.281,-178.992,6.170,148.814
C04907=1177.675,95.437,-51.263,-178.995,6.169,148.815
C04908=1177.681,95.188,-51.245,-178.997,6.168,148.815
C04909=1177.686,94.939,-51.227,-179.000,6.166,148.816
C04910=1177.691,94.689,-51.209,-179.002,6.166,148.816
C04911=1177.695,94.439,-51.190,-179.006,6.164,148.817
C04912=1177.700,94.190,-51.172,-179.008,6.163,148.817
C04913=1177.705,93.941,-51.154,-179.011,6.162,148.818
C04914=1177.710,93.692,-51.137,-179.014,6.160,148.818
C04915=1177.715,93.443,-51.119,-179.016,6.159,148.819
C04916=1177.719,93.194,-51.101,-179.019,6.158,148.819
C04917=1177.724,92.944,-51.083,-179.021,6.157,148.820
C04918=1177.729,92.695,-51.064,-179.024,6.156,148.820
C04919=1177.734,92.445,-51.046,-179.026,6.155,148.821
C04920=1177.739,92.196,-51.029,-179.029,6.153,148.821
C04921=1177.744,91.946,-51.011,-179.032,6.153,148.822
C04922=1177.749,91.697,-50.993,-179.034,6.151,148.822
C04923=1177.754,91.448,-50.975,-179.037,6.150,148.823
C04924=1177.758,91.199,-50.957,-179.040,6.149,148.823
C04925=1177.763,90.950,-50.939,-179.042,6.148,148.824
C04926=1177.768,90.701,-50.921,-179.045,6.146,148.824
C04927=1177.773,90.451,-50.903,-179.047,6.145,148.825
C04928=1177.778,90.201,-50.885,-179.050,6.144,148.825
C04929=1177.783,89.952,-50.868,-179.053,6.143,148.826
C04930=1177.788,89.702,-50.850,-179.056,6.142,148.827
C04931=1177.793,89.453,-50.832,-179.059,6.140,148.827
C04932=1177.797,89.204,-50.814,-179.061,6.139,148.827
C04933=1177.803,88.954,-50.796,-179.064,6.138,148.828
C04934=1177.807,88.705,-50.779,-179.066,6.137,148.828
C04935=1177.812,88.456,-50.761,-179.069,6.136,148.829
C04936=1177.817,88.207,-50.743,-179.071,6.135,148.830
C04937=1177.822,87.958,-50.725,-179.075,6.133,148.830
C04938=1177.827,87.708,-50.708,-179.077,6.132,148.831
C04939=1177.832,87.459,-50.690,-179.079,6.131,148.831
C04940=1177.837,87.210,-50.672,-179.082,6.130,148.832
C04941=1177.842,86.960,-50.655,-179.085,6.128,148.832
C04942=1177.846,86.711,-50.637,-179.087,6.128,148.833
C04943=1177.851,86.462,-50.619,-179.090,6.126,148.833
C04944=1177.856,86.212,-50.602,-179.093,6.126,148.834
C04945=1177.861,85.963,-50.584,-179.095,6.124,148.834
C04946=1177.866,85.714,-50.566,-179.098,6.123,148.835
C04947=1177.871,85.464,-50.549,-179.101,6.122,148.835
C04948=1177.875,85.215,-50.531,-179.103,6.121,148.836
C04949=1177.880,84.966,-50.513,-179.106,6.119,148.836
C04950=1177.886,84.716,-50.496,-179.108,6.119,148.837
C04951=1177.890,84.467,-50.478,-179.111,6.118,148.837
C04952=1177.895,84.218,-50.460,-179.114,6.116,148.838
C04953=1177.900,83.968,-50.443,-179.116,6.116,148.839
C04954=1177.905,83.719,-50.425,-179.119,6.114,148.839
C04955=1177.910,83.469,-50.408,-179.122,6.114,148.840
C04956=1177.915,83.220,-50.390,-179.124,6.112,148.840
C04957=1177.920,82.970,-50.373,-179.126,6.111,148.840
C04958=1177.924,82.722,-50.356,-179.130,6.110,148.841
C04959=1177.929,82.472,-50.338,-179.132,6.109,148.842
C04960=1177.934,82.223,-50.320,-179.135,6.107,148.842
C04961=1177.939,81.974,-50.303,-179.137,6.106,148.843
C04962=1177.944,81.725,-50.286,-179.140,6.105,148.843
C04963=1177.949,81.475,-50.268,-179.143,6.104,148.844
C04964=1177.954,81.226,-50.251,-179.146,6.103,148.844
C04965=1177.959,80.977,-50.233,-179.148,6.102,148.845
C04966=1177.964,80.708,-50.215,-179.151,6.101,148.845
C04967=1177.969,80.439,-50.196,-179.153,6.100,148.846
C04968=1177.975,80.171,-50.177,-179.156,6.098,148.846
C04969=1177.980,79.903,-50.159,-179.160,6.097,148.847
C04970=1177.985,79.653,-50.142,-179.162,6.096,148.848
C04971=1177.990,79.404,-50.124,-179.165,6.095,148.848
C04972=1177.994,79.154,-50.107,-179.167,6.094,148.849
C04973=1177.999,78.905,-50.089,-179.170,6.093,148.849
C04974=1178.005,78.655,-50.072,-179.173,6.092,148.850
C04975=1178.010,78.407,-50.055,-179.175,6.091,148.850
C04976=1178.015,78.158,-50.037,-179.178,6.089,148.851
C04977=1178.020,77.908,-50.020,-179.180,6.089,148.851
C04978=1178.024,77.658,-50.003,-179.183,6.087,148.852
C04979=1178.029,77.409,-49.985,-179.186,6.087,148.853
C04980=1178.034,77.160,-49.969,-179.189,6.085,148.853
C04981=1178.039,76.911,-49.952,-179.191,6.084,148.853
C04982=1178.044,76.661,-49.934,-179.193,6.084,148.854
C04983=1178.049,76.412,-49.917,-179.196,6.082,148.854
C04984=1178.054,76.162,-49.900,-179.199,6.081,148.855
C04985=1178.058,75.913,-49.883,-179.201,6.080,148.856
C04986=1178.063,75.663,-49.865,-179.204,6.079,148.856
C04987=1178.069,75.415,-49.849,-179.207,6.077,148.857
C04988=1178.074,75.165,-49.832,-179.209,6.077,148.857
C04989=1178.079,74.916,-49.814,-179.212,6.076,148.858
C04990=1178.083,74.666,-49.797,-179.215,6.075,148.858
C04991=1178.088,74.416,-49.780,-179.217,6.074,148.859
C04992=1178.093,74.168,-49.764,-179.220,6.072,148.859
C04993=1178.098,73.918,-49.746,-179.222,6.071,148.860
C04994=1178.103,73.669,-49.729,-179.225,6.071,148.861
C04995=1178.108,73.419,-49.712,-179.228,6.069,148.861
C04996=1178.113,73.170,-49.695,-179.230,6.069,148.862
C04997=1178.118,72.921,-49.678,-179.233,6.067,148.862
C04998=1178.123,72.671,-49.661,-179.236,6.066,148.863
C04999=1178.128,72.422,-49.643,-179.238,6.065,148.863
C05000=1178.132,72.172,-49.627,-179.241,6.064,148.864
C05001=1178.138,71.923,-49.610,-179.243,6.063,148.864
C05002=1178.142,71.674,-49.593,-179.246,6.062,148.865
C05003=1178.147,71.424,-49.577,-179.248,6.061,148.865
C05004=1178.152,71.175,-49.559,-179.252,6.060,148.866
C05005=1178.157,70.926,-49.543,-179.254,6.059,148.866
C05006=1178.162,70.676,-49.526,-179.256,6.058,148.867
C05007=1178.167,70.426,-49.509,-179.259,6.057,148.867
C05008=1178.172,70.177,-49.491,-179.262,6.056,148.868
C05009=1178.177,69.929,-49.475,-179.265,6.054,148.869
C05010=1178.181,69.679,-49.458,-179.267,6.054,148.869
C05011=1178.187,69.429,-49.441,-179.269,6.053,148.870
C05012=1178.192,69.180,-49.425,-179.273,6.052,148.870
C05013=1178.197,68.931,-49.407,-179.275,6.051,148.871
C05014=1178.201,68.681,-49.391,-179.277,6.050,148.871
C05015=1178.206,68.432,-49.374,-179.280,6.049,148.872
C05016=1178.212,68.183,-49.357,-179.283,6.048,148.873
C05017=1178.216,67.933,-49.340,-179.285,6.046,148.873
C05018=1178.221,67.684,-49.324,-179.288,6.046,148.874
C05019=1178.227,67.435,-49.307,-179.291,6.045,148.874
C05020=1178.231,67.185,-49.290,-179.293,6.044,148.875
C05021=1178.235,66.936,-49.273,-179.296,6.043,148.875
C05022=1178.241,66.686,-49.257,-179.298,6.042,148.876
C05023=1178.246,66.436,-49.241,-179.301,6.041,148.876
C05024=1178.251,66.187,-49.224,-179.304,6.040,148.877
C05025=1178.256,65.938,-49.207,-179.307,6.039,148.878
C05026=1178.261,65.688,-49.190,-179.309,6.038,148.878
C05027=1178.265,65.439,-49.174,-179.312,6.037,148.879
C05028=1178.270,65.190,-49.157,-179.314,6.036,148.879
C05029=1178.276,64.940,-49.140,-179.317,6.035,148.880
C05030=1178.280,64.691,-49.123,-179.319,6.034,148.880
C05031=1178.285,64.442,-49.107,-179.322,6.033,148.881
C05032=1178.291,64.192,-49.091,-179.324,6.032,148.881
C05033=1178.295,63.942,-49.074,-179.327,6.031,148.882
C05034=1178.300,63.693,-49.058,-179.330,6.030,148.882
C05035=1178.305,63.444,-49.041,-179.332,6.029,148.883
C05036=1178.311,63.195,-49.024,-179.335,6.028,148.883
C05037=1178.315,62.945,-49.008,-179.338,6.027,148.884
C05038=1178.320,62.695,-48.991,-179.340,6.026,148.885
C05039=1178.325,62.446,-48.975,-179.343,6.025,148.885
C05040=1178.329,62.197,-48.958,-179.346,6.024,148.886
C05041=1178.335,61.948,-48.942,-179.348,6.023,148.886
C05042=1178.340,61.698,-48.926,-179.351,6.022,148.887
C05043=1178.344,61.448,-48.909,-179.353,6.021,148.887
C05044=1178.350,61.199,-48.893,-179.356,6.021,148.888
C05045=1178.354,60.949,-48.877,-179.359,6.019,148.888
C05046=1178.360,60.700,-48.860,-179.361,6.018,148.889
C05047=1178.365,60.451,-48.843,-179.363,6.018,148.890
C05048=1178.370,60.202,-48.827,-179.367,6.016,148.890
C05049=1178.375,59.952,-48.811,-179.369,6.016,148.891
C05050=1178.380,59.703,-48.795,-179.371,6.015,148.891
C05051=1178.384,59.454,-48.778,-179.375,6.013,148.892
C05052=1178.389,59.203,-48.762,-179.377,6.013,148.892
C05053=1178.395,58.954,-48.745,-179.379,6.012,148.893
C05054=1178.399,58.705,-48.728,-179.382,6.010,148.894
C05055=1178.405,58.455,-48.713,-179.385,6.010,148.894
C05056=1178.409,58.206,-48.696,-179.387,6.009,148.895
C05057=1178.414,57.957,-48.681,-179.390,6.008,148.895
C05058=1178.419,57.707,-48.664,-179.392,6.007,148.896
C05059=1178.424,57.458,-48.648,-179.395,6.006,148.896
C05060=1178.429,57.208,-48.632,-179.398,6.006,148.897
C05061=1178.434,56.959,-48.615,-179.400,6.004,148.898
C05062=1178.439,56.709,-48.599,-179.403,6.004,148.898
C05063=1178.444,56.461,-48.583,-179.405,6.003,148.899
C05064=1178.449,56.210,-48.566,-179.408,6.001,148.899
C05065=1178.454,55.961,-48.550,-179.410,6.000,148.900
C05066=1178.459,55.711,-48.534,-179.413,6.000,148.900
C05067=1178.464,55.462,-48.518,-179.416,5.999,148.901
C05068=1178.469,55.212,-48.502,-179.418,5.998,148.902
C05069=1178.474,54.964,-48.486,-179.421,5.997,148.902
C05070=1178.480,54.695,-48.469,-179.424,5.996,148.903
C05071=1178.485,54.426,-48.451,-179.426,5.995,148.903
C05072=1178.490,54.158,-48.434,-179.430,5.994,148.904
C05073=1178.495,53.890,-48.417,-179.432,5.993,148.905
C05074=1178.500,53.639,-48.401,-179.434,5.992,148.905
C05075=1178.505,53.391,-48.384,-179.438,5.991,148.906
C05076=1178.511,53.141,-48.369,-179.440,5.990,148.906
C05077=1178.515,52.892,-48.352,-179.443,5.990,148.907
C05078=1178.521,52.642,-48.336,-179.445,5.989,148.907
C05079=1178.525,52.392,-48.320,-179.448,5.987,148.908
C05080=1178.530,52.144,-48.304,-179.451,5.987,148.909
C05081=1178.535,51.893,-48.288,-179.453,5.986,148.909
C05082=1178.540,51.645,-48.272,-179.456,5.985,148.910
C05083=1178.546,51.395,-48.256,-179.458,5.984,148.910
C05084=1178.550,51.145,-48.240,-179.461,5.983,148.911
C05085=1178.555,50.897,-48.225,-179.463,5.983,148.911
C05086=1178.560,50.647,-48.209,-179.466,5.981,148.912
C05087=1178.565,50.397,-48.193,-179.469,5.981,148.913
C05088=1178.570,50.148,-48.177,-179.471,5.980,148.913
C05089=1178.575,49.898,-48.161,-179.474,5.978,148.914
C05090=1178.580,49.649,-48.145,-179.476,5.978,148.914
C05091=1178.585,49.399,-48.129,-179.479,5.977,148.915
C05092=1178.590,49.150,-48.113,-179.482,5.977,148.915
C05093=1178.595,48.901,-48.097,-179.484,5.975,148.916
C05094=1178.599,48.651,-48.081,-179.487,5.974,148.917
C05095=1178.605,48.402,-48.066,-179.489,5.973,148.917
C05096=1178.610,48.153,-48.050,-179.492,5.973,148.918
C05097=1178.615,47.902,-48.034,-179.495,5.972,148.918
C05098=1178.620,47.653,-48.019,-179.497,5.971,148.919
C05099=1178.625,47.404,-48.002,-179.500,5.970,148.919
C05100=1178.629,47.155,-47.987,-179.502,5.969,148.920
C05101=1178.635,46.905,-47.971,-179.505,5.968,148.921
C05102=1178.640,46.656,-47.956,-179.508,5.968,148.921
C05103=1178.645,46.406,-47.939,-179.510,5.967,148.922
C05104=1178.650,46.157,-47.924,-179.512,5.966,148.922
C05105=1178.655,45.908,-47.909,-179.515,5.964,148.923
C05106=1178.659,45.658,-47.893,-179.518,5.964,148.923
C05107=1178.665,45.408,-47.877,-179.521,5.963,148.924
C05108=1178.670,45.159,-47.861,-179.523,5.963,148.925
C05109=1178.675,44.909,-47.845,-179.526,5.961,148.925
C05110=1178.679,44.660,-47.830,-179.528,5.960,148.926
C05111=1178.685,44.411,-47.814,-179.531,5.960,148.926
C05112=1178.689,44.161,-47.798,-179.533,5.959,148.927
C05113=1178.695,43.911,-47.783,-179.536,5.958,148.927
C05114=1178.699,43.662,-47.768,-179.539,5.957,148.928
C05115=1178.705,43.413,-47.752,-179.541,5.956,148.929
C05116=1178.710,43.163,-47.736,-179.544,5.956,148.929
C05117=1178.714,42.914,-47.721,-179.546,5.955,148.930
C05118=1178.720,42.664,-47.705,-179.549,5.954,148.930
C05119=1178.725,42.415,-47.690,-179.552,5.953,148.931
C05120=1178.730,42.165,-47.674,-179.554,5.952,148.932
C05121=1178.734,41.916,-47.659,-179.556,5.952,148.932
C05122=1178.740,41.666,-47.643,-179.560,5.950,148.933
C05123=1178.745,41.417,-47.628,-179.562,5.950,148.933
C05124=1178.749,41.167,-47.612,-179.564,5.949,148.934
C05125=1178.755,40.918,-47.597,-179.567,5.948,148.934
C05126=1178.760,40.668,-47.581,-179.569,5.948,148.935
C05127=1178.765,40.419,-47.566,-179.572,5.946,148.936
C05128=1178.770,40.169,-47.550,-179.575,5.946,148.936
C05129=1178.775,39.920,-47.535,-179.577,5.945,148.937
C05130=1178.780,39.671,-47.520,-179.579,5.944,148.937
C05131=1178.785,39.421,-47.504,-179.582,5.944,148.938
C05132=1178.790,39.172,-47.489,-179.585,5.942,148.939
C05133=1178.794,38.922,-47.473,-179.587,5.941,148.939
C05134=1178.800,38.673,-47.458,-179.590,5.941,148.940
C05135=1178.804,38.423,-47.443,-179.592,5.940,148.940
C05136=1178.810,38.174,-47.427,-179.595,5.940,148.941
C05137=1178.815,37.925,-47.411,-179.598,5.938,148.942
C05138=1178.820,37.674,-47.397,-179.600,5.937,148.942
C05139=1178.825,37.425,-47.381,-179.603,5.937,148.943
C05140=1178.830,37.176,-47.366,-179.605,5.936,148.943
C05141=1178.835,36.926,-47.351,-179.608,5.936,148.944
C05142=1178.840,36.677,-47.335,-179.611,5.934,148.944
C05143=1178.845,36.428,-47.320,-179.613,5.933,148.945
C05144=1178.850,36.177,-47.305,-179.616,5.933,148.946
C05145=1178.855,35.928,-47.290,-179.618,5.932,148.946
C05146=1178.860,35.679,-47.274,-179.620,5.932,148.947
C05147=1178.865,35.430,-47.259,-179.624,5.930,148.947
C05148=1178.870,35.180,-47.244,-179.626,5.929,148.948
C05149=1178.875,34.930,-47.229,-179.628,5.929,148.949
C05150=1178.880,34.681,-47.214,-179.631,5.928,148.949
C05151=1178.885,34.431,-47.198,-179.633,5.928,148.950
C05152=1178.890,34.182,-47.183,-179.636,5.927,148.950
C05153=1178.895,33.932,-47.169,-179.639,5.926,148.951
C05154=1178.900,33.683,-47.153,-179.641,5.925,148.951
C05155=1178.905,33.434,-47.138,-179.644,5.924,148.952
C05156=1178.910,33.184,-47.122,-179.646,5.923,148.953
C05157=1178.915,32.935,-47.108,-179.649,5.923,148.953
C05158=1178.921,32.685,-47.093,-179.651,5.923,148.954
C05159=1178.925,32.436,-47.078,-179.654,5.921,148.954
C05160=1178.930,32.185,-47.062,-179.657,5.920,148.955
C05161=1178.935,31.936,-47.047,-179.659,5.920,148.956
C05162=1178.940,31.687,-47.032,-179.662,5.919,148.956
C05163=1178.945,31.437,-47.017,-179.664,5.918,148.957
C05164=1178.950,31.188,-47.002,-179.667,5.918,148.958
C05165=1178.955,30.939,-46.987,-179.670,5.916,148.958
C05166=1178.960,30.689,-46.973,-179.672,5.916,148.959
C05167=1178.966,30.440,-46.957,-179.674,5.915,148.959
C05168=1178.970,30.190,-46.942,-179.677,5.914,148.960
C05169=1178.975,29.941,-46.928,-179.680,5.914,148.960
C05170=1178.981,29.691,-46.912,-179.682,5.913,148.961
C05171=1178.986,29.442,-46.898,-179.685,5.912,148.962
C05172=1178.991,29.192,-46.882,-179.688,5.911,148.962
C05173=1178.996,28.942,-46.868,-179.690,5.910,148.963
C05174=1179.001,28.674,-46.852,-179.693,5.910,148.963
C05175=1179.007,28.405,-46.835,-179.695,5.909,148.964
C05176=1179.012,28.136,-46.820,-179.698,5.908,148.965
C05177=1179.018,27.867,-46.803,-179.701,5.908,148.965
C05178=1179.023,27.618,-46.789,-179.703,5.907,148.966
C05179=1179.027,27.369,-46.774,-179.706,5.906,148.967
C05180=1179.033,27.118,-46.759,-179.709,5.906,148.967
C05181=1179.038,26.869,-46.744,-179.711,5.904,148.968
C05182=1179.043,26.620,-46.730,-179.714,5.904,148.968
C05183=1179.048,26.370,-46.714,-179.716,5.903,148.969
C05184=1179.053,26.121,-46.700,-179.719,5.902,148.970
C05185=1179.058,25.871,-46.685,-179.721,5.902,148.970
C05186=1179.063,25.622,-46.671,-179.724,5.901,148.971
C05187=1179.068,25.372,-46.655,-179.726,5.900,148.971
C05188=1179.073,25.123,-46.641,-179.729,5.899,148.972
C05189=1179.078,24.874,-46.626,-179.732,5.898,148.972
C05190=1179.083,24.624,-46.611,-179.734,5.898,148.973
C05191=1179.088,24.374,-46.597,-179.737,5.897,148.974
C05192=1179.093,24.125,-46.582,-179.739,5.897,148.974
C05193=1179.098,23.875,-46.567,-179.742,5.896,148.975
C05194=1179.103,23.626,-46.552,-179.744,5.896,148.976
C05195=1179.108,23.376,-46.538,-179.747,5.895,148.976
C05196=1179.113,23.126,-46.523,-179.749,5.894,148.977
C05197=1179.118,22.877,-46.508,-179.752,5.893,148.977
C05198=1179.123,22.627,-46.494,-179.755,5.892,148.978
C05199=1179.128,22.377,-46.479,-179.757,5.892,148.979
C05200=1179.133,22.128,-46.464,-179.759,5.891,148.979
C05201=1179.138,21.879,-46.450,-179.762,5.890,148.980
C05202=1179.143,21.629,-46.436,-179.765,5.890,148.980
C05203=1179.148,21.380,-46.421,-179.767,5.889,148.981
C05204=1179.154,21.130,-46.406,-179.769,5.888,148.982
C05205=1179.159,20.881,-46.392,-179.772,5.888,148.982
C05206=1179.163,20.632,-46.377,-179.775,5.886,148.983
C05207=1179.168,20.382,-46.363,-179.778,5.886,148.983
C05208=1179.173,20.132,-46.348,-179.780,5.885,148.984
C05209=1179.178,19.883,-46.334,-179.782,5.884,148.984
C05210=1179.184,19.633,-46.318,-179.785,5.884,148.985
C05211=1179.189,19.383,-46.304,-179.788,5.883,148.986
C05212=1179.194,19.134,-46.290,-179.790,5.883,148.986
C05213=1179.199,18.885,-46.276,-179.792,5.882,148.987
C05214=1179.204,18.635,-46.262,-179.795,5.882,148.988
C05215=1179.209,18.386,-46.247,-179.797,5.881,148.988
C05216=1179.214,18.136,-46.232,-179.800,5.880,148.989
C05217=1179.219,17.886,-46.218,-179.803,5.879,148.989
C05218=1179.224,17.636,-46.203,-179.805,5.878,148.990
C05219=1179.229,17.387,-46.189,-179.808,5.878,148.991
C05220=1179.235,17.138,-46.174,-179.811,5.877,148.991
C05221=1179.240,16.889,-46.160,-179.813,5.876,148.992
C05222=1179.245,16.639,-46.146,-179.815,5.876,148.992
C05223=1179.249,16.389,-46.132,-179.818,5.875,148.993
C05224=1179.254,16.140,-46.117,-179.820,5.874,148.994
C05225=1179.259,15.890,-46.103,-179.823,5.874,148.994
C05226=1179.264,15.640,-46.089,-179.826,5.874,148.995
C05227=1179.270,15.391,-46.075,-179.828,5.873,148.995
C05228=1179.275,15.142,-46.060,-179.830,5.872,148.996
C05229=1179.280,14.892,-46.045,-179.833,5.872,148.997
C05230=1179.284,14.643,-46.031,-179.835,5.871,148.997
C05231=1179.289,14.393,-46.017,-179.838,5.870,148.998
C05232=1179.295,14.144,-46.003,-179.841,5.869,148.999
C05233=1179.300,13.894,-45.989,-179.843,5.868,148.999
C05234=1179.305,13.644,-45.974,-179.846,5.868,149.000
C05235=1179.310,13.395,-45.960,-179.849,5.867,149.000
C05236=1179.315,13.145,-45.946,-179.851,5.866,149.001
C05237=1179.320,12.896,-45.932,-179.853,5.866,149.002
C05238=1179.325,12.646,-45.918,-179.856,5.865,149.002
C05239=1179.330,12.397,-45.903,-179.858,5.865,149.003
C05240=1179.335,12.147,-45.889,-179.861,5.864,149.003
C05241=1179.341,11.898,-45.875,-179.863,5.864,149.004
C05242=1179.346,11.648,-45.861,-179.866,5.863,149.004
C05243=1179.351,11.398,-45.847,-179.868,5.862,149.005
C05244=1179.356,11.149,-45.832,-179.871,5.862,149.006
C05245=1179.361,10.900,-45.819,-179.873,5.861,149.006
C05246=1179.366,10.650,-45.804,-179.876,5.861,149.007
C05247=1179.371,10.400,-45.790,-179.878,5.860,149.008
C05248=1179.376,10.151,-45.776,-179.881,5.859,149.008
C05249=1179.382,9.902,-45.762,-179.883,5.859,149.009
C05250=1179.387,9.651,-45.748,-179.886,5.857,149.010
C05251=1179.391,9.402,-45.735,-179.889,5.857,149.010
C05252=1179.396,9.152,-45.720,-179.891,5.856,149.011
C05253=1179.402,8.903,-45.706,-179.894,5.856,149.011
C05254=1179.407,8.653,-45.692,-179.896,5.855,149.012
C05255=1179.412,8.404,-45.678,-179.899,5.854,149.012
C05256=1179.416,8.154,-45.664,-179.901,5.854,149.013
C05257=1179.422,7.905,-45.650,-179.904,5.853,149.014
C05258=1179.427,7.655,-45.636,-179.906,5.853,149.014
C05259=1179.432,7.405,-45.622,-179.909,5.852,149.015
C05260=1179.437,7.156,-45.608,-179.911,5.851,149.015
C05261=1179.442,6.907,-45.594,-179.914,5.851,149.016
C05262=1179.447,6.657,-45.580,-179.916,5.850,149.017
C05263=1179.453,6.407,-45.567,-179.918,5.849,149.017
C05264=1179.458,6.157,-45.552,-179.921,5.849,149.018
C05265=1179.462,5.908,-45.539,-179.924,5.848,149.019
C05266=1179.468,5.659,-45.525,-179.926,5.848,149.019
C05267=1179.473,5.409,-45.511,-179.929,5.847,149.020
C05268=1179.478,5.159,-45.497,-179.931,5.847,149.021
C05269=1179.483,4.910,-45.483,-179.934,5.846,149.021
C05270=1179.488,4.661,-45.469,-179.936,5.845,149.022
C05271=1179.492,4.411,-45.455,-179.939,5.845,149.022
C05272=1179.498,4.161,-45.442,-179.941,5.844,149.023
C05273=1179.503,3.912,-45.428,-179.944,5.844,149.023
C05274=1179.508,3.662,-45.413,-179.946,5.843,149.024
C05275=1179.513,3.413,-45.401,-179.949,5.843,149.025
C05276=1179.518,3.163,-45.386,-179.951,5.842,149.025
C05277=1179.523,2.913,-45.372,-179.954,5.841,149.026
C05278=1179.529,2.644,-45.358,-179.956,5.841,149.027
C05279=1179.535,2.375,-45.343,-179.959,5.840,149.027
C05280=1179.539,2.106,-45.328,-179.962,5.839,149.028
C05281=1179.545,1.836,-45.313,-179.965,5.839,149.029
C05282=1179.551,1.587,-45.300,-179.967,5.838,149.029
C05283=1179.556,1.337,-45.286,-179.970,5.837,149.030
C05284=1179.561,1.088,-45.272,-179.972,5.837,149.031
C05285=1179.566,0.838,-45.259,-179.975,5.836,149.031
C05286=1179.571,0.588,-45.245,-179.977,5.835,149.032
C05287=1179.577,0.339,-45.231,-179.980,5.835,149.032
C05288=1179.581,0.089,-45.218,-179.982,5.834,149.033
C05289=1179.587,-0.160,-45.205,-179.985,5.834,149.034
C05290=1179.592,-0.410,-45.190,-179.987,5.833,149.034
C05291=1179.596,-0.659,-45.177,-179.989,5.832,149.035
C05292=1179.602,-0.909,-45.163,-179.992,5.832,149.035
C05293=1179.607,-1.159,-45.149,-179.995,5.831,149.036
C05294=1179.612,-1.408,-45.136,-179.997,5.831,149.037
C05295=1179.617,-1.658,-45.122,-180.000,5.830,149.037
C05296=1179.623,-1.907,-45.109,179.998,5.830,149.038
C05297=1179.627,-2.157,-45.095,179.996,5.830,149.038
C05298=1179.633,-2.406,-45.082,179.993,5.829,149.039
C05299=1179.637,-2.656,-45.068,179.991,5.829,149.040
C05300=1179.643,-2.905,-45.055,179.988,5.828,149.040
C05301=1179.648,-3.155,-45.041,179.986,5.827,149.041
C05302=1179.652,-3.405,-45.028,179.983,5.827,149.042
C05303=1179.658,-3.654,-45.014,179.981,5.826,149.042
C05304=1179.662,-3.904,-45.001,179.979,5.826,149.043
C05305=1179.668,-4.153,-44.987,179.976,5.825,149.043
C05306=1179.673,-4.404,-44.974,179.973,5.825,149.044
C05307=1179.678,-4.652,-44.960,179.971,5.824,149.045
C05308=1179.683,-4.903,-44.947,179.968,5.823,149.045
C05309=1179.688,-5.152,-44.934,179.966,5.823,149.046
C05310=1179.693,-5.402,-44.920,179.964,5.822,149.046
C05311=1179.698,-5.651,-44.907,179.961,5.822,149.047
C05312=1179.703,-5.901,-44.893,179.958,5.821,149.048
C05313=1179.709,-6.150,-44.880,179.956,5.820,149.048
C05314=1179.714,-6.400,-44.867,179.953,5.820,149.049
C05315=1179.719,-6.649,-44.853,179.951,5.819,149.050
C05316=1179.724,-6.899,-44.840,179.948,5.819,149.050
C05317=1179.730,-7.149,-44.827,179.946,5.818,149.051
C05318=1179.735,-7.398,-44.813,179.943,5.818,149.052
C05319=1179.740,-7.648,-44.800,179.941,5.817,149.052
C05320=1179.745,-7.897,-44.787,179.938,5.816,149.053
C05321=1179.750,-8.147,-44.773,179.936,5.816,149.053
C05322=1179.755,-8.396,-44.760,179.934,5.816,149.054
C05323=1179.760,-8.646,-44.747,179.932,5.815,149.055
C05324=1179.765,-8.895,-44.734,179.929,5.815,149.055
C05325=1179.770,-9.145,-44.721,179.926,5.814,149.056
C05326=1179.775,-9.395,-44.707,179.924,5.814,149.056
C05327=1179.780,-9.645,-44.694,179.921,5.813,149.057
C05328=1179.786,-9.894,-44.681,179.919,5.813,149.058
C05329=1179.791,-10.143,-44.668,179.916,5.812,149.058
C05330=1179.796,-10.394,-44.654,179.914,5.811,149.059
C05331=1179.801,-10.643,-44.642,179.911,5.811,149.060
C05332=1179.805,-10.892,-44.628,179.909,5.810,149.060
C05333=1179.811,-11.142,-44.615,179.906,5.810,149.061
C05334=1179.816,-11.392,-44.602,179.904,5.809,149.061
C05335=1179.822,-11.642,-44.589,179.901,5.809,149.062
C05336=1179.826,-11.890,-44.575,179.899,5.808,149.063
C05337=1179.832,-12.141,-44.562,179.896,5.807,149.063
C05338=1179.837,-12.390,-44.549,179.894,5.808,149.064
C05339=1179.841,-12.640,-44.536,179.892,5.807,149.064
C05340=1179.847,-12.890,-44.523,179.889,5.806,149.065
C05341=1179.852,-13.139,-44.510,179.887,5.806,149.066
C05342=1179.856,-13.388,-44.497,179.884,5.806,149.067
C05343=1179.862,-13.638,-44.484,179.882,5.805,149.067
C05344=1179.867,-13.887,-44.471,179.879,5.804,149.068
C05345=1179.873,-14.138,-44.457,179.877,5.804,149.068
C05346=1179.878,-14.387,-44.445,179.874,5.803,149.069
C05347=1179.882,-14.637,-44.432,179.872,5.803,149.070
C05348=1179.888,-14.887,-44.419,179.869,5.802,149.070
C05349=1179.893,-15.136,-44.406,179.867,5.801,149.071
C05350=1179.898,-15.385,-44.392,179.865,5.802,149.071
C05351=1179.903,-15.635,-44.379,179.862,5.801,149.072
C05352=1179.909,-15.884,-44.367,179.860,5.800,149.073
C05353=1179.913,-16.134,-44.354,179.857,5.800,149.073
C05354=1179.918,-16.384,-44.341,179.855,5.799,149.074
C05355=1179.924,-16.633,-44.328,179.852,5.799,149.075
C05356=1179.929,-16.883,-44.315,179.850,5.798,149.075
C05357=1179.934,-17.133,-44.302,179.847,5.798,149.076
C05358=1179.940,-17.382,-44.289,179.845,5.797,149.077
C05359=1179.944,-17.632,-44.276,179.842,5.796,149.077
C05360=1179.949,-17.881,-44.263,179.840,5.797,149.078
C05361=1179.954,-18.131,-44.251,179.838,5.796,149.078
C05362=1179.960,-18.380,-44.238,179.835,5.795,149.079
C05363=1179.965,-18.630,-44.225,179.833,5.795,149.080
C05364=1179.970,-18.880,-44.212,179.830,5.795,149.080
C05365=1179.975,-19.129,-44.200,179.828,5.794,149.081
C05366=1179.980,-19.379,-44.186,179.825,5.793,149.081
C05367=1179.985,-19.629,-44.173,179.823,5.793,149.082
C05368=1179.990,-19.878,-44.161,179.820,5.792,149.083
C05369=1179.996,-20.127,-44.148,179.818,5.792,149.083
C05370=1180.001,-20.378,-44.135,179.816,5.792,149.084
C05371=1180.006,-20.628,-44.123,179.813,5.791,149.085
C05372=1180.011,-20.877,-44.110,179.811,5.791,149.085
C05373=1180.016,-21.126,-44.098,179.808,5.790,149.086
C05374=1180.021,-21.376,-44.085,179.806,5.790,149.087
C05375=1180.027,-21.626,-44.071,179.803,5.789,149.087
C05376=1180.032,-21.875,-44.059,179.801,5.788,149.088
C05377=1180.037,-22.125,-44.046,179.798,5.788,149.088
C05378=1180.042,-22.375,-44.033,179.797,5.788,149.089
C05379=1180.047,-22.624,-44.021,179.794,5.787,149.090
C05380=1180.053,-22.874,-44.008,179.791,5.787,149.090
C05381=1180.058,-23.123,-43.995,179.789,5.787,149.091
C05382=1180.063,-23.393,-43.982,179.786,5.786,149.091
C05383=1180.069,-23.663,-43.968,179.784,5.785,149.092
C05384=1180.074,-23.932,-43.954,179.781,5.785,149.093
C05385=1180.080,-24.203,-43.941,179.778,5.784,149.093
C05386=1180.085,-24.452,-43.929,179.776,5.784,149.094
C05387=1180.091,-24.702,-43.915,179.773,5.783,149.095
C05388=1180.095,-24.952,-43.902,179.771,5.783,149.095
C05389=1180.100,-25.201,-43.890,179.768,5.782,149.096
C05390=1180.106,-25.451,-43.878,179.766,5.783,149.097
C05391=1180.111,-25.700,-43.865,179.764,5.782,149.097
C05392=1180.116,-25.949,-43.853,179.761,5.781,149.098
C05393=1180.121,-26.199,-43.840,179.759,5.781,149.099
C05394=1180.126,-26.449,-43.828,179.756,5.780,149.099
C05395=1180.131,-26.699,-43.815,179.754,5.780,149.100
C05396=1180.136,-26.948,-43.803,179.751,5.779,149.100
C05397=1180.141,-27.197,-43.790,179.749,5.779,149.101
C05398=1180.146,-27.448,-43.778,179.747,5.779,149.102
C05399=1180.151,-27.697,-43.765,179.744,5.778,149.102
C05400=1180.156,-27.947,-43.753,179.742,5.778,149.103
C05401=1180.162,-28.197,-43.741,179.739,5.777,149.103
C05402=1180.168,-28.446,-43.728,179.737,5.776,149.104
C05403=1180.173,-28.696,-43.715,179.734,5.776,149.105
C05404=1180.178,-28.945,-43.703,179.732,5.776,149.105
C05405=1180.183,-29.195,-43.690,179.730,5.776,149.106
C05406=1180.188,-29.445,-43.678,179.727,5.775,149.107
C05407=1180.193,-29.695,-43.666,179.725,5.774,149.107
C05408=1180.198,-29.944,-43.653,179.722,5.774,149.108
C05409=1180.204,-30.194,-43.641,179.720,5.773,149.109
C05410=1180.209,-30.443,-43.629,179.718,5.774,149.109
C05411=1180.214,-30.693,-43.616,179.715,5.773,149.110
C05412=1180.219,-30.943,-43.604,179.713,5.772,149.110
C05413=1180.224,-31.193,-43.591,179.710,5.772,149.111
C05414=1180.229,-31.442,-43.580,179.708,5.771,149.112
C05415=1180.234,-31.692,-43.567,179.705,5.771,149.112
C05416=1180.239,-31.941,-43.555,179.703,5.771,149.113
C05417=1180.244,-32.191,-43.543,179.701,5.770,149.114
C05418=1180.250,-32.440,-43.530,179.698,5.770,149.114
C05419=1180.255,-32.690,-43.518,179.696,5.769,149.115
C05420=1180.260,-32.939,-43.506,179.693,5.769,149.115
C05421=1180.266,-33.189,-43.494,179.691,5.768,149.116
C05422=1180.271,-33.439,-43.481,179.689,5.769,149.117
C05423=1180.276,-33.689,-43.469,179.687,5.768,149.117
C05424=1180.281,-33.939,-43.456,179.684,5.767,149.118
C05425=1180.286,-34.189,-43.444,179.681,5.767,149.119
C05426=1180.291,-34.438,-43.432,179.679,5.766,149.119
C05427=1180.297,-34.688,-43.420,179.677,5.766,149.120
C05428=1180.301,-34.937,-43.408,179.674,5.766,149.121
C05429=1180.306,-35.187,-43.396,179.672,5.765,149.121
C05430=1180.312,-35.436,-43.383,179.669,5.765,149.122
C05431=1180.317,-35.686,-43.372,179.667,5.764,149.122
C05432=1180.322,-35.935,-43.359,179.664,5.764,149.123
C05433=1180.328,-36.185,-43.347,179.663,5.764,149.124
C05434=1180.333,-36.435,-43.335,179.660,5.763,149.124
C05435=1180.338,-36.684,-43.323,179.657,5.763,149.125
C05436=1180.343,-36.934,-43.311,179.655,5.762,149.125
C05437=1180.348,-37.183,-43.299,179.652,5.762,149.126
C05438=1180.353,-37.433,-43.287,179.650,5.762,149.127
C05439=1180.358,-37.683,-43.274,179.648,5.761,149.127
C05440=1180.364,-37.933,-43.262,179.645,5.761,149.128
C05441=1180.369,-38.183,-43.250,179.643,5.760,149.129
C05442=1180.374,-38.432,-43.238,179.640,5.760,149.129
C05443=1180.379,-38.681,-43.227,179.639,5.760,149.130
C05444=1180.385,-38.931,-43.215,179.636,5.759,149.131
C05445=1180.390,-39.181,-43.202,179.633,5.759,149.131
C05446=1180.395,-39.431,-43.190,179.631,5.758,149.132
C05447=1180.401,-39.681,-43.178,179.628,5.758,149.132
C05448=1180.405,-39.930,-43.166,179.626,5.758,149.133
C05449=1180.410,-40.180,-43.154,179.624,5.757,149.134
C05450=1180.416,-40.429,-43.143,179.621,5.757,149.134
C05451=1180.421,-40.679,-43.130,179.619,5.756,149.135
C05452=1180.426,-40.928,-43.119,179.617,5.756,149.136
C05453=1180.431,-41.178,-43.107,179.615,5.756,149.136
C05454=1180.436,-41.428,-43.095,179.612,5.755,149.137
C05455=1180.442,-41.678,-43.082,179.610,5.755,149.137
C05456=1180.446,-41.927,-43.071,179.607,5.754,149.138
C05457=1180.452,-42.177,-43.059,179.605,5.755,149.139
C05458=1180.457,-42.427,-43.047,179.602,5.754,149.139
C05459=1180.462,-42.676,-43.035,179.600,5.753,149.140
C05460=1180.467,-42.926,-43.023,179.597,5.753,149.141
C05461=1180.472,-43.176,-43.011,179.595,5.752,149.141
C05462=1180.478,-43.426,-43.000,179.593,5.752,149.142
C05463=1180.483,-43.674,-42.988,179.591,5.752,149.143
C05464=1180.488,-43.924,-42.976,179.588,5.752,149.143
C05465=1180.494,-44.174,-42.964,179.586,5.751,149.144
C05466=1180.498,-44.424,-42.953,179.584,5.751,149.144
C05467=1180.504,-44.674,-42.941,179.581,5.751,149.145
C05468=1180.509,-44.923,-42.928,179.579,5.750,149.146
C05469=1180.514,-45.173,-42.917,179.576,5.749,149.146
C05470=1180.519,-45.423,-42.905,179.573,5.749,149.147
C05471=1180.524,-45.672,-42.893,179.572,5.749,149.147
C05472=1180.529,-45.922,-42.882,179.569,5.749,149.148
C05473=1180.535,-46.172,-42.870,179.567,5.748,149.149
C05474=1180.541,-46.421,-42.859,179.564,5.747,149.149
C05475=1180.545,-46.670,-42.847,179.562,5.748,149.150
C05476=1180.550,-46.920,-42.835,179.560,5.747,149.151
C05477=1180.556,-47.170,-42.823,179.557,5.746,149.151
C05478=1180.561,-47.420,-42.812,179.555,5.746,149.152
C05479=1180.566,-47.670,-42.800,179.553,5.746,149.153
C05480=1180.571,-47.920,-42.788,179.550,5.746,149.153
C05481=1180.576,-48.169,-42.777,179.548,5.745,149.154
C05482=1180.582,-48.419,-42.765,179.545,5.745,149.155
C05483=1180.587,-48.668,-42.754,179.544,5.745,149.155
C05484=1180.592,-48.918,-42.742,179.541,5.744,149.156
C05485=1180.598,-49.168,-42.730,179.538,5.744,149.156
C05486=1180.603,-49.438,-42.717,179.536,5.743,149.157
C05487=1180.609,-49.708,-42.704,179.533,5.743,149.158
C05488=1180.614,-49.979,-42.693,179.531,5.742,149.158
